// TIA Portal V18 program export: 1 tag tables, 8 data types, 17 data blocks, 20 code blocks (in call order from the OBs), 0 instance data blocks

VAR_GLOBAL   // PLC tag table "Default tag table"
   "AI11.01.01" AT %IW64 : Int;   // AHU NF Перепад тиску повітря (2.40)
   "AI11.01.02" AT %IW66 : Int;   // HS Вихід нагрівача (10.11)
   "DI11.01.01" AT %I0.0 : Bool;   // HS Режим роботи "Зима"
   "DI11.01.02" AT %I0.1 : Bool;   // HS Режим роботи "Авто"
   "DI11.01.03" AT %I0.2 : Bool;   // HS Відмова Котел 1
   "DI11.01.04" AT %I0.3 : Bool;   // HS Відмова Котел 2
   "DI11.01.05" AT %I0.4 : Bool;   // HS Норм. рівень води Котел 1 (10.80)
   "DI11.01.06" AT %I0.5 : Bool;   // HS Низький тиск Котел 1 (10.71)
   "DI11.01.07" AT %I0.6 : Bool;   // HS Високий тиск Котел 1 (10.72)
   "DI11.01.08" AT %I0.7 : Bool;   // HS Норм. рівень води Котел 2 (10.81)
   "DI11.01.09" AT %I1.0 : Bool;   // HS Низький тиск Котел 1 (10.73)
   "DI11.01.10" AT %I1.1 : Bool;   // HS Високий тиск Котел 1 (10.74)
   "DI11.01.11" AT %I1.2 : Bool;
   "DI11.01.12" AT %I1.3 : Bool;
   "DI11.01.13" AT %I1.4 : Bool;
   "DI11.01.14" AT %I1.5 : Bool;
   "DO11.01.01" AT %Q0.0 : Bool;
   "DO11.01.02" AT %Q0.1 : Bool;
   "DO11.01.03" AT %Q0.2 : Bool;
   "DO11.01.04" AT %Q0.3 : Bool;
   "DO11.01.05" AT %Q0.4 : Bool;
   "DO11.01.06" AT %Q0.5 : Bool;
   "DO11.01.07" AT %Q0.6 : Bool;
   "DO11.01.08" AT %Q0.7 : Bool;
   "DO11.01.09" AT %Q1.0 : Bool;
   "DO11.01.10" AT %Q1.1 : Bool;
   "AI11.02.01" AT %IW68 : Int;
   "AI11.02.02" AT %IW70 : Int;
   "AI11.02.03" AT %IW72 : Int;
   "AI11.02.04" AT %IW74 : Int;
   "AI11.02.05" AT %IW76 : Int;
   "AI11.02.06" AT %IW78 : Int;
   "AI11.02.07" AT %IW80 : Int;
   "AI11.02.08" AT %IW82 : Int;
   "AO11.03.01" AT %QW64 : Int;
   "AO11.03.02" AT %QW66 : Int;
   "AO11.03.03" AT %QW68 : Int;
   "AO11.03.04" AT %QW70 : Int;
   "DI11.04.01" AT %I2.0 : Bool;
   "DI11.04.02" AT %I2.1 : Bool;
   "DI11.04.03" AT %I2.2 : Bool;
   "DI11.04.04" AT %I2.3 : Bool;
   "DI11.04.05" AT %I2.4 : Bool;
   "DI11.04.06" AT %I2.5 : Bool;
   "DI11.04.07" AT %I2.6 : Bool;
   "DI11.04.08" AT %I2.7 : Bool;
   "DI11.04.09" AT %I3.0 : Bool;
   "DI11.04.10" AT %I3.1 : Bool;
   "DI11.04.11" AT %I3.2 : Bool;
   "DI11.04.12" AT %I3.3 : Bool;
   "DI11.04.13" AT %I3.4 : Bool;
   "DI11.04.14" AT %I3.5 : Bool;
   "DI11.04.15" AT %I3.6 : Bool;
   "DI11.04.16" AT %I3.7 : Bool;
   "DI11.05.01" AT %I4.0 : Bool;
   "DI11.05.02" AT %I4.1 : Bool;
   "DI11.05.03" AT %I4.2 : Bool;
   "DI11.05.04" AT %I4.3 : Bool;
   "DI11.05.05" AT %I4.4 : Bool;
   "DI11.05.06" AT %I4.5 : Bool;
   "DI11.05.07" AT %I4.6 : Bool;
   "DI11.05.08" AT %I4.7 : Bool;
   "DI11.05.09" AT %I5.0 : Bool;
   "DI11.05.10" AT %I5.1 : Bool;
   "DI11.05.11" AT %I5.2 : Bool;
   "DI11.05.12" AT %I5.3 : Bool;
   "DI11.05.13" AT %I5.4 : Bool;
   "DI11.05.14" AT %I5.5 : Bool;
   "DI11.05.15" AT %I5.6 : Bool;
   "DI11.05.16" AT %I5.7 : Bool;
   "DI11.06.01" AT %I6.0 : Bool;
   "DI11.06.02" AT %I6.1 : Bool;
   "DI11.06.03" AT %I6.2 : Bool;
   "DI11.06.04" AT %I6.3 : Bool;
   "DI11.06.05" AT %I6.4 : Bool;
   "DI11.06.06" AT %I6.5 : Bool;
   "DI11.06.07" AT %I6.6 : Bool;
   "DI11.06.08" AT %I6.7 : Bool;
   "DI11.06.09" AT %I7.0 : Bool;
   "DI11.06.10" AT %I7.1 : Bool;
   "DI11.06.11" AT %I7.2 : Bool;
   "DI11.06.12" AT %I7.3 : Bool;
   "DI11.06.13" AT %I7.4 : Bool;
   "DI11.06.14" AT %I7.5 : Bool;
   "DI11.06.15" AT %I7.6 : Bool;
   "DI11.06.16" AT %I7.7 : Bool;
   "DI11.07.01" AT %I8.0 : Bool;
   "DI11.07.02" AT %I8.1 : Bool;
   "DI11.07.03" AT %I8.2 : Bool;
   "DI11.07.04" AT %I8.3 : Bool;
   "DI11.07.05" AT %I8.4 : Bool;
   "DI11.07.06" AT %I8.5 : Bool;
   "DI11.07.07" AT %I8.6 : Bool;
   "DI11.07.08" AT %I8.7 : Bool;
   "DI11.07.09" AT %I9.0 : Bool;
   "DI11.07.10" AT %I9.1 : Bool;
   "DI11.07.11" AT %I9.2 : Bool;
   "DI11.07.12" AT %I9.3 : Bool;
   "DI11.07.13" AT %I9.4 : Bool;
   "DI11.07.14" AT %I9.5 : Bool;
   "DI11.07.15" AT %I9.6 : Bool;
   "DI11.07.16" AT %I9.7 : Bool;
   "DO11.08.01" AT %Q2.0 : Bool;
   "DO11.08.02" AT %Q2.1 : Bool;
   "DO11.08.03" AT %Q2.2 : Bool;
   "DO11.08.04" AT %Q2.3 : Bool;
   "DO11.08.05" AT %Q2.4 : Bool;
   "DO11.08.06" AT %Q2.5 : Bool;
   "DO11.08.07" AT %Q2.6 : Bool;
   "DO11.08.08" AT %Q2.7 : Bool;
   "DO11.08.09" AT %Q3.0 : Bool;
   "DO11.08.10" AT %Q3.1 : Bool;
   "DO11.08.11" AT %Q3.2 : Bool;
   "DO11.08.12" AT %Q3.3 : Bool;
   "DO11.08.13" AT %Q3.4 : Bool;
   "DO11.08.14" AT %Q3.5 : Bool;
   "DO11.08.15" AT %Q3.6 : Bool;
   "DO11.08.16" AT %Q3.7 : Bool;
   "DO11.09.01" AT %Q4.0 : Bool;
   "DO11.09.02" AT %Q4.1 : Bool;
   "DO11.09.03" AT %Q4.2 : Bool;
   "DO11.09.04" AT %Q4.3 : Bool;
   "DO11.09.05" AT %Q4.4 : Bool;
   "DO11.09.06" AT %Q4.5 : Bool;
   "DO11.09.07" AT %Q4.6 : Bool;
   "DO11.09.08" AT %Q4.7 : Bool;
   "DO11.09.09" AT %Q5.0 : Bool;
   "DO11.09.10" AT %Q5.1 : Bool;
   "DO11.09.11" AT %Q5.2 : Bool;
   "DO11.09.12" AT %Q5.3 : Bool;
   "DO11.09.13" AT %Q5.4 : Bool;
   "DO11.09.14" AT %Q5.5 : Bool;
   "DO11.09.15" AT %Q5.6 : Bool;
   "DO11.09.16" AT %Q5.7 : Bool;
   "AI11.10.01" AT %IW84 : Int;
   "AI11.10.02" AT %IW86 : Int;
   "AI11.10.03" AT %IW88 : Int;
   "AI11.10.04" AT %IW90 : Int;
   "AI11.10.05" AT %IW92 : Int;
   "AI11.10.06" AT %IW94 : Int;
   "AI11.10.07" AT %IW96 : Int;
   "AI11.10.08" AT %IW98 : Int;
   "AO11.11.01" AT %QW72 : Int;
   "AO11.11.02" AT %QW74 : Int;
   "AO11.11.03" AT %QW76 : Int;
   "AO11.11.04" AT %QW78 : Int;
END_VAR

TYPE "UDT_HWModulesMap"
// stored: IsFailsafeCompliant false
   STRUCT
      cRack : Byte;
      cModule : Byte;
      wLaddr1 : Word;
      wLaddr2 : Word;
      iDiagBuffer : USInt;
      iOwnState : UInt;
      wMaintenanceState : DWord;
      wComponentStateDetail : DWord;
      iOperatingState : UInt;
   END_STRUCT;
END_TYPE

TYPE "UDT_VirtModulesMap"
// stored: IsFailsafeCompliant false
   STRUCT
      cRack : Byte;
      cModule : Byte;
      iDiagBuffer : USInt;
      iOwnState : UInt;
   END_STRUCT;
END_TYPE

TYPE "UDT_AIadv"
// stored: IsFailsafeCompliant false
   STRUCT
      rValue : Real;   // Real value
      rMin : Real;   // Scale Min
      rMax : Real;   // Scale Max
      rCalibration : Real;
      iFuncSystemID : Byte := 0;
      iFuncVar : Byte := 0;
      rFilterSet : Real;   // Filter value
   END_STRUCT;
END_TYPE

TYPE "UDT_DIadv"
// stored: IsFailsafeCompliant false
   STRUCT
      xInput : Bool;
      xMemoryIn : Bool;   // Temp
      xMemoryOut : Bool;
      xInversion : Bool;   // DIs label for monitoring
      xOutput : Bool;   // Filtered value
      xtemp1 : Bool;
      xtemp2 : Bool;
      xtemp3 : Bool;
      cMemory : Byte := 0;
      iCounterOut : Int;
      iCounterIn : Int;   // Counter for DIs EDGE
      cFuncSystemID : Byte := 0;
      cFuncVar : Byte := 0;
      cDelayOnSec : Byte := 0;   // Temp
      cDelayOffSec : Byte := 0;   // Temp
   END_STRUCT;
END_TYPE

TYPE "UDT_RTDadv"
// stored: IsFailsafeCompliant false
   STRUCT
      rValue : Real;   // Real value
      rFilterSet : Real;   // Filter value
      rCalibration : Real;   // Scale Min
      rDiv : Real := 100.0;   // Scale Max
      cFuncSystemID : Byte := 0;
      cFuncVar : Byte := 0;
      iReserv : Int;
   END_STRUCT;
END_TYPE

TYPE "UDT_vAO"
// stored: IsFailsafeCompliant false
   STRUCT
      rInput : Real;   // Value for AO
      cMOA : Byte := 0;   // Mode Manual/Off/Auto
      cFuncSystemID : Byte := 0;
      cFuncVar : Byte := 0;
      cMemory : Byte := 0;
      rManOutput : Real;   // Manual output
      iOutput : Int;   // Output for DAC
   END_STRUCT;
END_TYPE

TYPE "UDT_vDI"
// stored: IsFailsafeCompliant false
   STRUCT
      xInput : Bool;
      xMemoryIn : Bool;   // Temp
      xMemoryOut : Bool;
      xInversion : Bool;   // DIs label for monitoring
      xOutput : Bool;   // Filtered value
      xtemp1 : Bool;
      xtemp2 : Bool;
      xtemp3 : Bool;
      cMemory : Byte := 0;
      iCounterOut : Int;
      iCounterIn : Int;   // Counter for DIs EDGE
      cFuncSystemID : Byte := 0;
      cFuncVar : Byte := 0;
      cDelayOnSec : Byte := 0;   // Temp
      cDelayOffSec : Byte := 0;   // Temp
   END_STRUCT;
END_TYPE

TYPE "UDT_vDO"
// stored: IsFailsafeCompliant false
   STRUCT
      xInput : Bool;   // Value for DO
      xOutput : Bool;   // Phisicl output
      xMemoryIn : Bool;   // Internal
      xInversion : Bool;
      xMemoryOut : Bool;
      xReserv3 : Bool;
      xReserv4 : Bool;
      xReserv5 : Bool;
      iCounterIn : Int;   // Counter
      iCounterOut : Int;
      iFuncSystemID : Byte := 0;
      iFuncVar : Byte := 0;
      cMOA : Byte;   // Mode Manual/Off/Auto
      cMemory : Byte;
   END_STRUCT;
END_TYPE

DATA_BLOCK "ActualHWAlarmsList"   // DB10001
{ S7_Optimized_Access := 'FALSE' }
VERSION : 0.1
// stored: AutoNumber false, DBAccessibleFromOPCUA true, IsOnlyStoredInLoadMemory false, IsWriteProtectedInAS false
   VAR
      iActiveFaults : DInt;
      iWriteIndex : Int;
      Log { S7_SetPoint := 'True'} : Array[0..99] of "UDT_HWAlarmEntry";
   END_VAR
BEGIN
END_DATA_BLOCK

DATA_BLOCK "HWModulesConf"   // DB10002
{ S7_Optimized_Access := 'TRUE' }
VERSION : 0.1
// stored: AutoNumber false, DBAccessibleFromOPCUA true, IsOnlyStoredInLoadMemory false, IsRetainMemResEnabled false, IsWriteProtectedInAS false, MemoryReserve 100
   VAR
      HW { S7_SetPoint := 'True'} : Array[1..14] of "UDT_HWModulesMap";
   END_VAR
BEGIN
   HW[1..8].cRack := 11;
   HW[9..14].cRack := 12;
   HW[1].cModule := 1;
   HW[2].cModule := 2;
   HW[3].cModule := 3;
   HW[4].cModule := 4;
   HW[5].cModule := 5;
   HW[6].cModule := 6;
   HW[7..8].cModule := 7;
   HW[9].cModule := 0;
   HW[10].cModule := 1;
   HW[11].cModule := 2;
   HW[12].cModule := 3;
   HW[13].cModule := 4;
   HW[14].cModule := 5;
   HW[1].wLaddr1 := 263;
   HW[2].wLaddr1 := 269;
   HW[3].wLaddr1 := 270;
   HW[4].wLaddr1 := 286;
   HW[5].wLaddr1 := 271;
   HW[6].wLaddr1 := 272;
   HW[7].wLaddr1 := 287;
   HW[8].wLaddr1 := 288;
   HW[9].wLaddr1 := 280;
   HW[10].wLaddr1 := 282;
   HW[11].wLaddr1 := 283;
   HW[12].wLaddr1 := 284;
   HW[13].wLaddr1 := 285;
   HW[14].wLaddr1 := 281;
   HW[1].wLaddr2 := 264;
END_DATA_BLOCK

DATA_BLOCK "HeatingPLC_vAO_Vars"   // DB11002
{ S7_Optimized_Access := 'FALSE' }
VERSION : 0.1
// stored: AutoNumber false, DBAccessibleFromOPCUA true, IsOnlyStoredInLoadMemory false, IsWriteProtectedInAS false
   VAR
      vAO1 { S7_SetPoint := 'True'} : "UDT_vAO";
      vAO2 { S7_SetPoint := 'True'} : "UDT_vAO";
      vAO3 { S7_SetPoint := 'True'} : "UDT_vAO";
      vAO4 { S7_SetPoint := 'True'} : "UDT_vAO";
      vAO5 { S7_SetPoint := 'True'} : "UDT_vAO";
      vAO6 { S7_SetPoint := 'True'} : "UDT_vAO";
      vAO7 { S7_SetPoint := 'True'} : "UDT_vAO";
      vAO8 { S7_SetPoint := 'True'} : "UDT_vAO";
   END_VAR
BEGIN
END_DATA_BLOCK

DATA_BLOCK "HeatingPLC_vDO_Vars"   // DB11004
{ S7_Optimized_Access := 'FALSE' }
VERSION : 0.1
// stored: AutoNumber false, DBAccessibleFromOPCUA true, IsOnlyStoredInLoadMemory false, IsWriteProtectedInAS false
   VAR
      vDO1 { S7_SetPoint := 'True'} : "UDT_vDO";
      vDO2 { S7_SetPoint := 'True'} : "UDT_vDO";
      vDO3 { S7_SetPoint := 'True'} : "UDT_vDO";
      vDO4 { S7_SetPoint := 'True'} : "UDT_vDO";
      vDO5 { S7_SetPoint := 'True'} : "UDT_vDO";
      vDO6 { S7_SetPoint := 'True'} : "UDT_vDO";
      vDO7 { S7_SetPoint := 'True'} : "UDT_vDO";
      vDO8 { S7_SetPoint := 'True'} : "UDT_vDO";
   END_VAR
BEGIN
END_DATA_BLOCK

DATA_BLOCK "SS1_710A1_8RTD_AI_Vars"   // DB11021
{ S7_Optimized_Access := 'FALSE' }
VERSION : 0.1
// stored: AutoNumber false, DBAccessibleFromOPCUA true, IsOnlyStoredInLoadMemory false, IsWriteProtectedInAS false
   VAR
      AI1 { S7_SetPoint := 'True'} : "UDT_RTDadv";   // Зовнішня температура (1.99)
      AI2 { S7_SetPoint := 'True'} : "UDT_RTDadv";   // AHU NF Темп. зв. теплоносія (2.57)
      AI3 { S7_SetPoint := 'True'} : "UDT_RTDadv";   // AHU NF Темп. припл. пов. (2.56)
      AI4 { S7_SetPoint := 'True'} : "UDT_RTDadv";   // AHU NF Кімнатна темп. (2.69)
      AI5 { S7_SetPoint := 'True'} : "UDT_RTDadv";   // HS Темп. под. теплоносія в колекторі (10.50)
      AI6 { S7_SetPoint := 'True'} : "UDT_RTDadv";   // Температура зв. теплоносія (8.66)
      AI7 { S7_SetPoint := 'True'} : "UDT_RTDadv";   // Темп. припл. пов. (8.68)
      AI8 { S7_SetPoint := 'True'} : "UDT_RTDadv";   // HS Темп. зв. теплоносія (10.92)
   END_VAR
BEGIN
   AI1.rValue := 26.03;
   AI1.rFilterSet := 0.0;
   AI1.rCalibration := 0.0;
   AI1.rDiv := 100.0;
   AI1.cFuncSystemID := 0;
   AI1.cFuncVar := 0;
   AI1.iReserv := 0;
   AI2.rValue := 3276.7;
   AI2.rFilterSet := 0.0;
   AI2.rCalibration := 0.0;
   AI2.rDiv := 10.0;
   AI2.cFuncSystemID := 2;
   AI2.cFuncVar := 0;
   AI2.iReserv := 0;
   AI3.rValue := 26.7;
   AI3.rFilterSet := 0.0;
   AI3.rCalibration := 0.0;
   AI3.rDiv := 100.0;
   AI3.cFuncSystemID := 16#01;
   AI3.cFuncVar := 16#04;
   AI3.iReserv := 0;
   AI4.rValue := 22.39;
   AI4.rFilterSet := 0.0;
   AI4.rCalibration := 0.0;
   AI4.rDiv := 100.0;
   AI4.cFuncSystemID := 16#03;
   AI4.cFuncVar := 16#04;
   AI4.iReserv := 0;
   AI5.rValue := 24.7;
   AI5.rFilterSet := 0.0;
   AI5.rCalibration := 0.0;
   AI5.rDiv := 10.0;
   AI5.cFuncSystemID := 16#0A;
   AI5.cFuncVar := 16#01;
   AI5.iReserv := 0;
   AI6.rValue := 61.78;
   AI6.rFilterSet := 0.0;
   AI6.rCalibration := 0.0;
   AI6.rDiv := 100.0;
   AI6.cFuncSystemID := 16#0E;
   AI6.cFuncVar := 16#01;
   AI6.iReserv := 0;
   AI7.rValue := 28.62;
   AI7.rFilterSet := 0.0;
   AI7.rCalibration := 0.0;
   AI7.rDiv := 100.0;
   AI7.cFuncSystemID := 16#0E;
   AI7.cFuncVar := 16#02;
   AI7.iReserv := 0;
   AI8.rValue := 21.31;
   AI8.rFilterSet := 0.0;
   AI8.rCalibration := 0.0;
   AI8.rDiv := 100.0;
   AI8.cFuncSystemID := 16#03;
   AI8.cFuncVar := 16#06;
   AI8.iReserv := 0;
END_DATA_BLOCK

DATA_BLOCK "SS1_730A1_4AO_AO_Vars"   // DB11041
{ S7_Optimized_Access := 'FALSE' }
VERSION : 0.1
// stored: AutoNumber false, DBAccessibleFromOPCUA true, IsOnlyStoredInLoadMemory false, IsWriteProtectedInAS false
   VAR
      AO1 { S7_SetPoint := 'True'} : "UDT_AOadv";   // AHU NF вихід нагрівача (2.58)
      AO2 { S7_SetPoint := 'True'} : "UDT_AOadv";   // AHU NF приточна/рециркуляційна заслінка (2.51/2.52)
      AO3 : "UDT_AOadv";   // Вихід нагрівача (8.67)
      AO4 : "UDT_AOadv";   // AHU NF витяжна заслінка (2.70)
   END_VAR
BEGIN
   AO1.cFuncSystemID := 1;
   AO1.cFuncVar := 2;
   AO2.cFuncSystemID := 1;
   AO2.cFuncVar := 3;
   AO3.cFuncSystemID := 3;
   AO3.cFuncVar := 2;
   AO4.cFuncSystemID := 1;
   AO4.cFuncVar := 4;
END_DATA_BLOCK

DATA_BLOCK "SS1_750A1_16DI_DI_Vars"   // DB11051
{ S7_Optimized_Access := 'FALSE' }
VERSION : 0.1
// stored: AutoNumber false, DBAccessibleFromOPCUA true, IsOnlyStoredInLoadMemory false, IsWriteProtectedInAS false
   VAR
      DI1 : "UDT_DIadv";   // Індикація живлення SS-1
      DI2 : "UDT_DIadv";   // HS Несправність системи опалення
      DI3 : "UDT_DIadv";   // HS Ін. 1- ст пальник К1
      DI4 : "UDT_DIadv";   // HS Ін. 2- ст пальник К1
      DI5 : "UDT_DIadv";   // Резерв
      DI6 : "UDT_DIadv";   // HS Аварія пальник К1
      DI7 : "UDT_DIadv";   // HS Ін. 1- ст пальник К2
      DI8 : "UDT_DIadv";   // HS Ін. 2- ст пальник К2
      DI9 { S7_SetPoint := 'True'} : "UDT_DIadv";   // HS Аварія пальник К2
      DI10 { S7_SetPoint := 'True'} : "UDT_DIadv";   // Резерв
      DI11 { S7_SetPoint := 'True'} : "UDT_DIadv";   // Резерв
      DI12 { S7_SetPoint := 'True'} : "UDT_DIadv";   // AHU NF Аварія ККБ
      DI13 { S7_SetPoint := 'True'} : "UDT_DIadv";   // AHU NF Ін. 1- ст. ККБ
      DI14 { S7_SetPoint := 'True'} : "UDT_DIadv";   // AHU NF Ін. 2- ст. ККБ
      DI15 { S7_SetPoint := 'True'} : "UDT_DIadv";   // Гот. роб. сист. обігр. дизельпроводу (10.211)
      DI16 { S7_SetPoint := 'True'} : "UDT_DIadv";   // AHU NF Гот. роб. обігр. пов. засл. (2.202)
   END_VAR
BEGIN
   DI3.cFuncSystemID := 10;
   DI3.cFuncVar := 25;
   DI4.cFuncSystemID := 10;
   DI4.cFuncVar := 26;
   DI5.cFuncSystemID := 10;
   DI5.cFuncVar := 27;
   DI6.cFuncSystemID := 100;
   DI6.cFuncVar := 11;
   DI7.cFuncSystemID := 100;
   DI7.cFuncVar := 12;
   DI8.cFuncSystemID := 10;
   DI8.cFuncVar := 24;
   DI9.cFuncSystemID := 10;
   DI9.cFuncVar := 22;
   DI10.xInversion := true;
   DI10.cFuncSystemID := 10;
   DI10.cFuncVar := 23;
   DI11.cFuncSystemID := 10;
   DI11.cFuncVar := 7;
   DI12.cFuncSystemID := 10;
   DI12.cFuncVar := 2;
   DI13.xInversion := true;
   DI13.cFuncSystemID := 10;
   DI13.cFuncVar := 3;
   DI14.cFuncSystemID := 10;
   DI14.cFuncVar := 5;
   DI15.xInversion := true;
   DI15.cFuncSystemID := 10;
   DI15.cFuncVar := 6;
END_DATA_BLOCK

DATA_BLOCK "SS1_754A1_16DI_DI_Vars"   // DB11061
{ S7_Optimized_Access := 'FALSE' }
VERSION : 0.1
// stored: AutoNumber false, DBAccessibleFromOPCUA true, IsOnlyStoredInLoadMemory false, IsWriteProtectedInAS false
   VAR
      DI1 : "UDT_DIadv";   // AHU NF Термостат загр. замерз. (2.50)
      DI2 : "UDT_DIadv";   // AHU NF Авто. режим пр. вент. (2.200)
      DI3 : "UDT_DIadv";   // AHU NF 1-шв. пр. вент. (2.200)
      DI4 : "UDT_DIadv";   // AHU NF 2-шв. пр. вент. (2.200)
      DI5 : "UDT_DIadv";   // AHU NF Тепл. реле. 1-шв. пр. вент. (2.200)
      DI6 : "UDT_DIadv";   // AHU NF Тепл. реле. 2-шв. пр. вент. (2.200)
      DI7 : "UDT_DIadv";   // AHU NF Несправність пр. вент. (2.200)
      DI8 : "UDT_DIadv";   // AHU NF Інд. сервісний вимикач. пр. вент. (2.200)
      DI9 { S7_SetPoint := 'True'} : "UDT_DIadv";   // AHU NF Несправність клиновий ркмінь пр. вент. (2.54)
      DI10 { S7_SetPoint := 'True'} : "UDT_DIadv";   // AHU NF Забруднення пр. фільтру (2.53)
      DI11 { S7_SetPoint := 'True'} : "UDT_DIadv";   // AHU NF Робота цирк. насос (2.201)
      DI12 { S7_SetPoint := 'True'} : "UDT_DIadv";   // AHU NF Авто режим цирк. насос (2.201)
      DI13 { S7_SetPoint := 'True'} : "UDT_DIadv";   // AHU NF Несправність цирк. насос (2.201)
      DI14 { S7_SetPoint := 'True'} : "UDT_DIadv";   // HS Робота вн. насос К1 (10.209)
      DI15 { S7_SetPoint := 'True'} : "UDT_DIadv";   // HS Перегрів вн. насос К1 (10.209) термоконтакт
      DI16 { S7_SetPoint := 'True'} : "UDT_DIadv";   // HS Робота вн. насос К2 (10.210)
   END_VAR
BEGIN
   DI1.cFuncSystemID := 100;
   DI1.cFuncVar := 1;
   DI2.cFuncSystemID := 100;
   DI2.cFuncVar := 3;
   DI5.cFuncSystemID := 100;
   DI5.cFuncVar := 5;
   DI6.cFuncSystemID := 100;
   DI6.cFuncVar := 6;
END_DATA_BLOCK

DATA_BLOCK "SS1_758A1_16DI_DI_Vars"   // DB11061
{ S7_Optimized_Access := 'FALSE' }
VERSION : 0.1
// stored: AutoNumber false, DBAccessibleFromOPCUA true, IsOnlyStoredInLoadMemory false, IsWriteProtectedInAS false
   VAR
      DI1 : "UDT_DIadv";   // HS Перегрів вн. наос К2 (10.20) термоконтакт
      DI2 : "UDT_DIadv";   // HS Авто режим насосів опалення (10.202+10.203)
      DI3 : "UDT_DIadv";   // HS Несправність насос опалення 1 (10.202)
      DI4 : "UDT_DIadv";   // HS Несправність насос опалення 2 (10.203)
      DI5 : "UDT_DIadv";   // Робота обігріву дизельпроводу
      DI6 : "UDT_DIadv";   // Резерв
      DI7 : "UDT_DIadv";   // Перегрів двигуна тепл. вентиляторів (8.215+8.216)
      DI8 : "UDT_DIadv";   // Робота тепл. вентиляторів (8.215+8.216)
      DI9 { S7_SetPoint := 'True'} : "UDT_DIadv";   // Термостат загр. замерз. (8.73)
      DI10 { S7_SetPoint := 'True'} : "UDT_DIadv";   // Термостат загр. замерз. (8.74)
      DI11 { S7_SetPoint := 'True'} : "UDT_DIadv";   // Несправність цирк. насос (8.217)
      DI12 { S7_SetPoint := 'True'} : "UDT_DIadv";   // Робота цирк. насос (8.217)
      DI13 { S7_SetPoint := 'True'} : "UDT_DIadv";   // Авто режим цирк. насос (8.217)
      DI14 { S7_SetPoint := 'True'} : "UDT_DIadv";   // Забруднення пр. фільтру (8.71)
      DI15 { S7_SetPoint := 'True'} : "UDT_DIadv";   // Забруднення пр. фільтру (8.72)
      DI16 { S7_SetPoint := 'True'} : "UDT_DIadv";   // HS Робота насосу опалення 1 (10.202)
   END_VAR
BEGIN
   DI1.cFuncSystemID := 100;
   DI1.cFuncVar := 1;
   DI2.cFuncSystemID := 100;
   DI2.cFuncVar := 3;
   DI5.cFuncSystemID := 100;
   DI5.cFuncVar := 5;
   DI6.cFuncSystemID := 100;
   DI6.cFuncVar := 6;
END_DATA_BLOCK

DATA_BLOCK "SS1_762A1_16DI_DI_Vars"   // DB11061
{ S7_Optimized_Access := 'FALSE' }
VERSION : 0.1
// stored: AutoNumber false, DBAccessibleFromOPCUA true, IsOnlyStoredInLoadMemory false, IsWriteProtectedInAS false
   VAR
      DI1 : "UDT_DIadv";   // HS Робота насосу опалення 2 (10.203)
      DI2 : "UDT_DIadv";   // Резерв
      DI3 : "UDT_DIadv";   // Резерв
      DI4 : "UDT_DIadv";   // Резерв
      DI5 : "UDT_DIadv";   // Резерв
      DI6 : "UDT_DIadv";   // Резерв
      DI7 : "UDT_DIadv";   // Резерв
      DI8 : "UDT_DIadv";   // Резерв
      DI9 { S7_SetPoint := 'True'} : "UDT_DIadv";   // Резерв
      DI10 { S7_SetPoint := 'True'} : "UDT_DIadv";   // Резерв
      DI11 { S7_SetPoint := 'True'} : "UDT_DIadv";   // Резерв
      DI12 { S7_SetPoint := 'True'} : "UDT_DIadv";   // Резерв
      DI13 { S7_SetPoint := 'True'} : "UDT_DIadv";   // Резерв
      DI14 { S7_SetPoint := 'True'} : "UDT_DIadv";   // Резерв
      DI15 { S7_SetPoint := 'True'} : "UDT_DIadv";   // Резерв
      DI16 { S7_SetPoint := 'True'} : "UDT_DIadv";   // Резерв
   END_VAR
BEGIN
   DI1.cFuncSystemID := 100;
   DI1.cFuncVar := 1;
   DI2.cFuncSystemID := 100;
   DI2.cFuncVar := 3;
   DI5.cFuncSystemID := 100;
   DI5.cFuncVar := 5;
   DI6.cFuncSystemID := 100;
   DI6.cFuncVar := 6;
END_DATA_BLOCK

DATA_BLOCK "SS1_770A1_16DO_DO_Vars"   // DB11072
{ S7_Optimized_Access := 'FALSE' }
VERSION : 0.1
// stored: AutoNumber false, DBAccessibleFromOPCUA true, IsOnlyStoredInLoadMemory false, IsWriteProtectedInAS false
   VAR
      DO1 { S7_SetPoint := 'True'} : "UDT_DOadv";   // Резерв
      DO2 { S7_SetPoint := 'True'} : "UDT_DOadv";   // Резерв
      DO3 { S7_SetPoint := 'True'} : "UDT_DOadv";   // Вкл. тепл. вент (8.x)
      DO4 { S7_SetPoint := 'True'} : "UDT_DOadv";   // HS Вкл. насос (10.203)
      DO5 { S7_SetPoint := 'True'} : "UDT_DOadv";   // HS Вкл. насос (10.202)
      DO6 { S7_SetPoint := 'True'} : "UDT_DOadv";   // HS Дозвіл на роботу пальник 1- ст. К1
      DO7 { S7_SetPoint := 'True'} : "UDT_DOadv";   // HS Дозвіл на роботу пальник 2- ст. К1
      DO8 { S7_SetPoint := 'True'} : "UDT_DOadv";   // AHU NF Вкл. цирк. насос (2.202)
      DO9 { S7_SetPoint := 'True'} : "UDT_DOadv";   // AHU NF Дозвіл на роботу 1- ст. ККБ
      DO10 { S7_SetPoint := 'True'} : "UDT_DOadv";   // AHU NF Дозвіл на роботу 2- ст. ККБ
      DO11 { S7_SetPoint := 'True'} : "UDT_DOadv";   // AHU NF Дозвіл на роботу 3- ст. ККБ
      DO12 { S7_SetPoint := 'True'} : "UDT_DOadv";   // AHU NF Дозвіл на роботу 4- ст. ККБ
      DO13 { S7_SetPoint := 'True'} : "UDT_DOadv";   // AHU NF Вкл. 1- шв. пр. вент. (2.200)
      DO14 { S7_SetPoint := 'True'} : "UDT_DOadv";   // AHU NF Вкл. 2- шв. пр. вент. (2.200)
      DO15 { S7_SetPoint := 'True'} : "UDT_DOadv";   // HS Дозвіл на роботу пальник 1- ст. К2
      DO16 { S7_SetPoint := 'True'} : "UDT_DOadv";   // HS Дозвіл на роботу пальник 2- ст. К2
   END_VAR
BEGIN
   DO1.iFuncSystemID := 10;
   DO1.iFuncVar := 10;
   DO2.iFuncSystemID := 10;
   DO2.iFuncVar := 11;
   DO3.iFuncSystemID := 10;
   DO3.iFuncVar := 12;
   DO4.iFuncSystemID := 100;
   DO4.iFuncVar := 1;
   DO5.iFuncSystemID := 100;
   DO5.iFuncVar := 5;
   DO6.iFuncSystemID := 100;
   DO6.iFuncVar := 3;
   DO7.iFuncSystemID := 10;
   DO7.iFuncVar := 5;
   DO8.iFuncSystemID := 10;
   DO8.iFuncVar := 6;
   DO9.iFuncSystemID := 10;
   DO9.iFuncVar := 13;
   DO14.iFuncSystemID := 1;
   DO14.iFuncVar := 1;
   DO14.cMOA := 1;
   DO15.iFuncSystemID := 1;
   DO16.iFuncSystemID := 1;
   DO16.iFuncVar := 3;
END_DATA_BLOCK

DATA_BLOCK "SS1_774A1_16DO_DO_Vars"   // DB11072
{ S7_Optimized_Access := 'FALSE' }
VERSION : 0.1
// stored: AutoNumber false, DBAccessibleFromOPCUA true, IsOnlyStoredInLoadMemory false, IsWriteProtectedInAS false
   VAR
      DO1 { S7_SetPoint := 'True'} : "UDT_DOadv";   // HS Вкл. вн. насос К1 (10.209)
      DO2 { S7_SetPoint := 'True'} : "UDT_DOadv";   // HS Вкл. вн. насос К2 (10.210)
      DO3 { S7_SetPoint := 'True'} : "UDT_DOadv";   // Резерв
      DO4 { S7_SetPoint := 'True'} : "UDT_DOadv";   // HS Дозвіл на роботу котлів
      DO5 { S7_SetPoint := 'True'} : "UDT_DOadv";   // AHU NF Вкл. обігріву пов. засл. (2.202)
      DO6 { S7_SetPoint := 'True'} : "UDT_DOadv";   // Вкл. обігріву дизельпровода (10.211)
      DO7 { S7_SetPoint := 'True'} : "UDT_DOadv";   // Вкл. системи кондиціювання (7.208 + 7.210)
      DO8 { S7_SetPoint := 'True'} : "UDT_DOadv";   // Вкл. тепл. вентилятор (8.215 + 8.216)
      DO9 { S7_SetPoint := 'True'} : "UDT_DOadv";   // Вкл. цирк. насос (8.217)
      DO10 { S7_SetPoint := 'True'} : "UDT_DOadv";   // Резерв
      DO11 { S7_SetPoint := 'True'} : "UDT_DOadv";   // Резерв
      DO12 { S7_SetPoint := 'True'} : "UDT_DOadv";   // Резерв
      DO13 { S7_SetPoint := 'True'} : "UDT_DOadv";   // Резерв
      DO14 { S7_SetPoint := 'True'} : "UDT_DOadv";   // Резерв
      DO15 { S7_SetPoint := 'True'} : "UDT_DOadv";   // Резерв
      DO16 { S7_SetPoint := 'True'} : "UDT_DOadv";   // Резерв
   END_VAR
BEGIN
   DO1.iFuncSystemID := 10;
   DO1.iFuncVar := 10;
   DO2.iFuncSystemID := 10;
   DO2.iFuncVar := 11;
   DO3.iFuncSystemID := 10;
   DO3.iFuncVar := 12;
   DO4.iFuncSystemID := 100;
   DO4.iFuncVar := 1;
   DO5.iFuncSystemID := 100;
   DO5.iFuncVar := 5;
   DO6.iFuncSystemID := 100;
   DO6.iFuncVar := 3;
   DO7.iFuncSystemID := 10;
   DO7.iFuncVar := 5;
   DO8.iFuncSystemID := 10;
   DO8.iFuncVar := 6;
   DO9.iFuncSystemID := 10;
   DO9.iFuncVar := 13;
   DO14.iFuncSystemID := 1;
   DO14.iFuncVar := 1;
   DO14.cMOA := 1;
   DO15.iFuncSystemID := 1;
   DO16.iFuncSystemID := 1;
   DO16.iFuncVar := 3;
END_DATA_BLOCK

DATA_BLOCK "SS1_780A1_8xAI_AI_Vars"   // DB11031
{ S7_Optimized_Access := 'FALSE' }
VERSION : 0.1
// stored: AutoNumber false, DBAccessibleFromOPCUA true, IsOnlyStoredInLoadMemory false, IsWriteProtectedInAS false
   VAR
      AI1 { S7_SetPoint := 'True'} : "UDT_AIadv";   // HS Температура в прим. котельні (10.02)
      AI2 { S7_SetPoint := 'True'} : "UDT_AIadv";   // 4-wire
      AI3 { S7_SetPoint := 'True'} : "UDT_AIadv";   // HS Температура зв. теплоносія (10.12)
      AI4 { S7_SetPoint := 'True'} : "UDT_AIadv";   // 4-wire
      AI5 { S7_SetPoint := 'True'} : "UDT_AIadv";   // HS Температура подачі теплоносія (10.13)
      AI6 { S7_SetPoint := 'True'} : "UDT_AIadv";   // 4-wire
      AI7 { S7_SetPoint := 'True'} : "UDT_AIadv";   // Резерв
      AI8 { S7_SetPoint := 'True'} : "UDT_AIadv";   // Резерв
   END_VAR
BEGIN
   AI1.rValue := 0.3255208;
   AI1.rMin := 0.0;
   AI1.rMax := 1000.0;
   AI1.rCalibration := 0.0;
   AI1.iFuncSystemID := 16#00;
   AI1.iFuncVar := 16#00;
   AI1.rFilterSet := 0.0;
   AI2.rValue := 1.808449;
   AI2.rMin := 0.0;
   AI2.rMax := 1000.0;
   AI2.rCalibration := 0.0;
   AI2.iFuncSystemID := 16#00;
   AI2.iFuncVar := 16#00;
   AI2.rFilterSet := 0.0;
   AI3.rValue := 3.616898E-05;
   AI3.rMin := 0.0;
   AI3.rMax := 0.0;
   AI3.rCalibration := 0.0;
   AI3.iFuncSystemID := 16#00;
   AI3.iFuncVar := 16#00;
   AI3.rFilterSet := 0.0;
   AI4.rValue := 0.0003255208;
   AI4.rMin := 0.0;
   AI4.rMax := 0.0;
   AI4.rCalibration := 0.0;
   AI4.iFuncSystemID := 16#00;
   AI4.iFuncVar := 16#00;
   AI4.rFilterSet := 0.0;
   AI5.rValue := 6.04022;
   AI5.rMin := 0.0;
   AI5.rMax := 1000.0;
   AI5.rCalibration := 0.0;
   AI5.iFuncSystemID := 16#01;
   AI5.iFuncVar := 16#0A;
   AI5.rFilterSet := 0.0;
   AI6.rValue := 17.15549;
   AI6.rMin := 0.0;
   AI6.rMax := 15.0;
   AI6.rCalibration := 0.0;
   AI6.iFuncSystemID := 16#01;
   AI6.iFuncVar := 16#07;
   AI6.rFilterSet := 0.0;
   AI7.rValue := 29.49942;
   AI7.rMin := 0.0;
   AI7.rMax := 100.0;
   AI7.rCalibration := 0.0;
   AI7.iFuncSystemID := 16#00;
   AI7.iFuncVar := 16#00;
   AI7.rFilterSet := 0.0;
   AI8.rValue := 0.07957176;
   AI8.rMin := 0.0;
   AI8.rMax := 100.0;
   AI8.rCalibration := 0.0;
   AI8.iFuncSystemID := 16#00;
   AI8.iFuncVar := 16#00;
   AI8.rFilterSet := 0.0;
END_DATA_BLOCK

DATA_BLOCK "SS1_784A1_4AO_AO_Vars"   // DB11041
{ S7_Optimized_Access := 'FALSE' }
VERSION : 0.1
// stored: AutoNumber false, DBAccessibleFromOPCUA true, IsOnlyStoredInLoadMemory false, IsWriteProtectedInAS false
   VAR
      AO1 { S7_SetPoint := 'True'} : "UDT_AOadv";   // HS Вихід нагрівача контуру опалення (10.11)
      AO2 { S7_SetPoint := 'True'} : "UDT_AOadv";   // Резерв
      AO3 : "UDT_AOadv";   // Резерв
      AO4 : "UDT_AOadv";   // Резерв
   END_VAR
BEGIN
   AO1.cFuncSystemID := 1;
   AO1.cFuncVar := 2;
   AO2.cFuncSystemID := 1;
   AO2.cFuncVar := 3;
   AO3.cFuncSystemID := 3;
   AO3.cFuncVar := 2;
   AO4.cFuncSystemID := 1;
   AO4.cFuncVar := 4;
END_DATA_BLOCK

DATA_BLOCK "SS1_CPU1214_AI_Vars"   // DB11011
{ S7_Optimized_Access := 'FALSE' }
VERSION : 0.1
// stored: AutoNumber false, DBAccessibleFromOPCUA true, IsOnlyStoredInLoadMemory false, IsWriteProtectedInAS false
   VAR
      AI1 { S7_SetPoint := 'True'} : "UDT_AIadv";   // AHU NF Перепад тиску повітря (2.40)
      AI2 { S7_SetPoint := 'True'} : "UDT_AIadv";   // HS Вихід нагрівача (10.11)
   END_VAR
BEGIN
   AI1.rValue := 368.9236;
   AI1.rMin := 0.0;
   AI1.rMax := 50000.0;
   AI1.rCalibration := 0.0;
   AI1.iFuncSystemID := 2;
   AI1.iFuncVar := 2;
   AI1.rFilterSet := 0.0;
   AI2.rValue := 0.0;
   AI2.rMin := 0.0;
   AI2.rMax := 0.0;
   AI2.rCalibration := 0.0;
   AI2.iFuncSystemID := 10;
   AI2.iFuncVar := 7;
   AI2.rFilterSet := 0.0;
END_DATA_BLOCK

DATA_BLOCK "SS1_CPU1214_DI_Vars"   // DB11013
{ S7_Optimized_Access := 'FALSE' }
VERSION : 0.1
// stored: AutoNumber false, DBAccessibleFromOPCUA true, IsOnlyStoredInLoadMemory false, IsWriteProtectedInAS false
   VAR
      DI1 : "UDT_DIadv";   // HS Режим роботи "Зима"
      DI2 : "UDT_DIadv";   // HS Режим роботи "Авто"
      DI3 : "UDT_DIadv";   // HS Відмова Котел 1
      DI4 : "UDT_DIadv";   // HS Відмова Котел 2
      DI5 : "UDT_DIadv";   // HS Норм. рівень води Котел 1 (10.80)
      DI6 : "UDT_DIadv";   // HS Низький тиск Котел 1 (10.71)
      DI7 { S7_SetPoint := 'True'} : "UDT_DIadv";   // HS Високий тиск Котел 1 (10.72)
      DI8 { S7_SetPoint := 'True'} : "UDT_DIadv";   // HS Норм. рівень води Котел 2 (10.81)
      DI9 { S7_SetPoint := 'True'} : "UDT_DIadv";   // HS Низький тиск Котел 1 (10.73)
      DI10 { S7_SetPoint := 'True'} : "UDT_DIadv";   // HS Високий тиск Котел 1 (10.74)
      DI11 { S7_SetPoint := 'True'} : "UDT_DIadv";   // Резерв
      DI12 { S7_SetPoint := 'True'} : "UDT_DIadv";   // Резерв
      DI13 { S7_SetPoint := 'True'} : "UDT_DIadv";   // Резерв
      DI14 { S7_SetPoint := 'True'} : "UDT_DIadv";   // Резерв
   END_VAR
BEGIN
   DI1.cFuncSystemID := 3;
   DI1.cFuncVar := 19;
   DI2.cFuncSystemID := 3;
   DI2.cFuncVar := 8;
   DI3.cFuncSystemID := 3;
   DI3.cFuncVar := 9;
   DI4.cFuncSystemID := 3;
   DI4.cFuncVar := 20;
   DI5.cFuncSystemID := 3;
   DI5.cFuncVar := 7;
   DI6.cFuncSystemID := 3;
   DI6.cFuncVar := 21;
   DI8.cFuncSystemID := 10;
   DI8.cFuncVar := 41;
   DI9.cFuncSystemID := 10;
   DI9.cFuncVar := 43;
   DI10.cFuncSystemID := 3;
   DI10.cFuncVar := 16;
   DI11.cFuncSystemID := 0;
   DI11.cFuncVar := 0;
   DI12.cFuncSystemID := 0;
   DI12.cFuncVar := 0;
   DI13.cFuncSystemID := 0;
   DI13.cFuncVar := 0;
END_DATA_BLOCK

DATA_BLOCK "SS1_CPU1214_DO_Vars"   // DB11014
{ S7_Optimized_Access := 'FALSE' }
VERSION : 0.1
// stored: AutoNumber false, DBAccessibleFromOPCUA true, IsOnlyStoredInLoadMemory false, IsWriteProtectedInAS false
   VAR
      DO1 { S7_SetPoint := 'True'} : "UDT_DOadv";   // Резерв
      DO2 { S7_SetPoint := 'True'} : "UDT_DOadv";   // Резерв
      DO3 { S7_SetPoint := 'True'} : "UDT_DOadv";   // Резерв
      DO4 { S7_SetPoint := 'True'} : "UDT_DOadv";   // Резерв
      DO5 { S7_SetPoint := 'True'} : "UDT_DOadv";   // Резерв
      DO6 : "UDT_DOadv";   // Резерв
      DO7 { S7_SetPoint := 'True'} : "UDT_DOadv";   // Резерв
      DO8 { S7_SetPoint := 'True'} : "UDT_DOadv";   // Резерв
      DO9 { S7_SetPoint := 'True'} : "UDT_DOadv";   // Резерв
      DO10 { S7_SetPoint := 'True'} : "UDT_DOadv";   // Резерв
   END_VAR
BEGIN
END_DATA_BLOCK

ORGANIZATION_BLOCK "Main"   // OB1, LAD, ProgramCycle
TITLE = "Main Program Sweep (Cycle)"
{ S7_Optimized_Access := 'TRUE' }
VERSION : 0.1
// stored: AutoNumber true, IsIECCheckEnabled false, SetENOAutomatically false
   VAR_INPUT
      Initial_Call : Bool;   // Initial call of this OB
      Remanence : Bool;   // =True, if remanent data are available
   END_VAR
BEGIN
END_ORGANIZATION_BLOCK

FUNCTION "AIadv" : Void   // FC10013, FBD
{ S7_Optimized_Access := 'TRUE' }
VERSION : 0.1
// stored: AutoNumber false, IsIECCheckEnabled false, SetENOAutomatically false, UDAEnableTagReadback false
   VAR_INPUT
      iInput : Int;
      rFilterValue : Real;
      rMin : Real;
      rMax : Real;
      rCalibration : Real;
   END_VAR
   VAR_OUTPUT
      rOutput : Real;
   END_VAR
   VAR_TEMP
      rNorm : Real;
      rScaled : Real;
      rOut_real : Real;
   END_VAR
   VAR CONSTANT
      iRawMin : Int := 0;
      iRawMax : Int := 27648;
   END_VAR
BEGIN

REGION Network 1 (SCL)
   #rNorm := NORM_X(
                    MIN := #iRawMin,
                    VALUE := #iInput,
                    MAX := #iRawMax);
END_REGION

REGION Network 2 (SCL)
   #rScaled := SCALE_X(
                       MIN := #rMin,
                       VALUE := #rNorm,
                       MAX := #rMax);
END_REGION

REGION Network 3 (SCL): // --- Обмеження межами ---
   IF #rScaled < #rMin THEN
       #rScaled := #rMin;
   ELSIF #rScaled > #rMax THEN
       #rScaled := #rMax;
   END_IF;
END_REGION

REGION Network 4 (SCL): // --- Калібрування (зсув) ---
   #rOutput := #rScaled + #rCalibration;
END_REGION

REGION Network 5 (SCL): // --- Підготовка коеф. фільтра ---
   // rFilterSet = 1.0 → фільтр «прозорий» (швидка реакція, без згладжування).
   // 
   // rFilterSet = 0.1…0.3 → м’яке згладжування.
   // 
   // rFilterSet = 0.0 → вихід «заморожений».
   // --- Підготовка коеф. фільтра ---
   //rAlpha := rFilterSet;/
   //IF rAlpha < 0.0 THEN
   //    rAlpha := 0.0;
   //END_IF;
   //IF rAlpha > 1.0 THEN
   //    rAlpha := 1.0;
   //END_IF;

   // --- Ініціалізація ---
   //IF xInit THEN
   //    rY := rScaledRaw;/
   //    xInit := FALSE;
   //END_IF;

   // --- Фільтр: y = y + α*(x - y) ---
   //rY := rY + rAlpha * (rScaledRaw - rY);

   // --- Вихід ---
   //#rOutput := rY;
END_REGION
END_FUNCTION

FUNCTION "AOadv" : Void   // FC10012, FBD
{ S7_Optimized_Access := 'TRUE' }
VERSION : 0.1
// stored: AutoNumber false, IsIECCheckEnabled false, SetENOAutomatically false, UDAEnableTagReadback false
   VAR_INPUT
      rInput : Real;   // 0 to 100
      cM0A : Byte;   // 0-direct / 1-reverse / 0-outp_off / 1- out=MAN_OUTPUT /2 -out=input
      rManOutput : Real;
   END_VAR
   VAR_OUTPUT
      iOutput : Int;
   END_VAR
   VAR_TEMP
      rOut : Real;
      rOutScaled : Real;
      rManOutputTemp : Real;
      iManOutputTemp : Int;
   END_VAR
   VAR CONSTANT
      iRawMin : Int := 0;
      iRawMax : Int := 27648;
   END_VAR
BEGIN

REGION Network 1 (SCL): // --- Вибір режиму ---
   // --- Вибір режиму ---
   CASE #cM0A OF
       0: // Off
           #rOut := 0.0;
       1: // Manual
           #rOut := #rManOutput;
       2: // Auto
           #rOut := #rInput;
       ELSE
           #rOut := 0.0; // захист від некоректних значень
   END_CASE;
END_REGION

REGION Network 2 (SCL): // --- Обмеження в межах 0.0…100.0 ---
   // --- Обмеження в межах 0.0…100.0 ---
   IF #rOut < 0.0 THEN
       #rOut := 0.0;
   ELSIF
       #rOut > 100.0 THEN
       #rOut := 100.0;
   END_IF;
END_REGION

REGION Network 3 (SCL)
   #rOutScaled := (#rOut * 27648.0) / 100;
END_REGION

REGION Network 4 (SCL)
   IF #rOutScaled < 0.0 THEN
       #rOutScaled := 0.0;
   ELSIF
       #rOutScaled > 27648.0 THEN
       #rOutScaled := 27648.0;
   END_IF;
END_REGION

REGION Network 5 (SCL)
   #iOutput := REAL_TO_INT(#rOutScaled + 0.5);
END_REGION
END_FUNCTION

FUNCTION "DOadv" : Void   // FC10009, LAD
{ S7_Optimized_Access := 'TRUE' }
VERSION : 0.1
// stored: AutoNumber false, IsIECCheckEnabled false, SetENOAutomatically false, UDAEnableTagReadback false
   VAR_INPUT
      xInput : Bool;
      xInversion : Bool;   // 0-direct / 1-reverse
      cMOA : Byte;
   END_VAR
   VAR_OUTPUT
      xOutput : Bool;
   END_VAR
   VAR_IN_OUT
      xMemoryOut : Bool;
      xMemoryIn : Bool;
      cMemory : Byte;
      iCounterIn : Int;
      iCounterOut : Int;
   END_VAR
   VAR_TEMP
      InOut_1 : Bool;
   END_VAR
BEGIN

REGION Network 1 (SCL)
   CASE #cMOA OF
       0: // OFF
           #xOutput := FALSE;

       1: // MANUAL
           #xOutput := TRUE;

       2: // AUTO
           #xOutput :=#xInput;

   ELSE
       #xOutput := FALSE;
   END_CASE;
END_REGION

REGION Network 2 (SCL)
   IF #xInversion THEN
       #xOutput := NOT #xOutput;
   END_IF;
END_REGION

REGION Network 3 (SCL)
   IF (#xMemoryIn XOR #xInput) THEN
       IF #iCounterIn > 30000 THEN
           #iCounterIn := 5;
       ELSE
           #iCounterIn := #iCounterIn + 1;
       END_IF;
   END_IF;
   #xMemoryIn := #xInput;
END_REGION

REGION Network 4 (SCL)
   IF (#xMemoryOut XOR #xOutput) THEN
       IF #iCounterOut > 30000 THEN
           #iCounterOut := 5;
       ELSE
           #iCounterOut := #iCounterOut + 1;
       END_IF;
   END_IF;
   #xMemoryOut := #xOutput;
END_REGION
END_FUNCTION

FUNCTION "DObasic" : Void   // FC10004, FBD
{ S7_Optimized_Access := 'TRUE' }
VERSION : 0.1
// stored: AutoNumber false, IsIECCheckEnabled false, SetENOAutomatically false, UDAEnableTagReadback false
   VAR_INPUT
      xInput : Bool;
      cM0A : Byte;   // 0-direct / 1-reverse / 0-outp_off / 1- aut=1 /2 -out=input
   END_VAR
   VAR_OUTPUT
      iCounter : Int;
      xOutput : Bool;
   END_VAR
   VAR_IN_OUT
      Bit_Count_1 : Bool;
   END_VAR
   VAR_TEMP
      cM0A_0 : Bool;
      cM0A_1 : Bool;
      cM0A_2 : Bool;
   END_VAR
   VAR CONSTANT
      bit_count : Bool;
   END_VAR
   VAR_TEMP   // added for the SCL form of the ladder/FBD networks
      _w1 : Bool;
   END_VAR
BEGIN

REGION Network 1
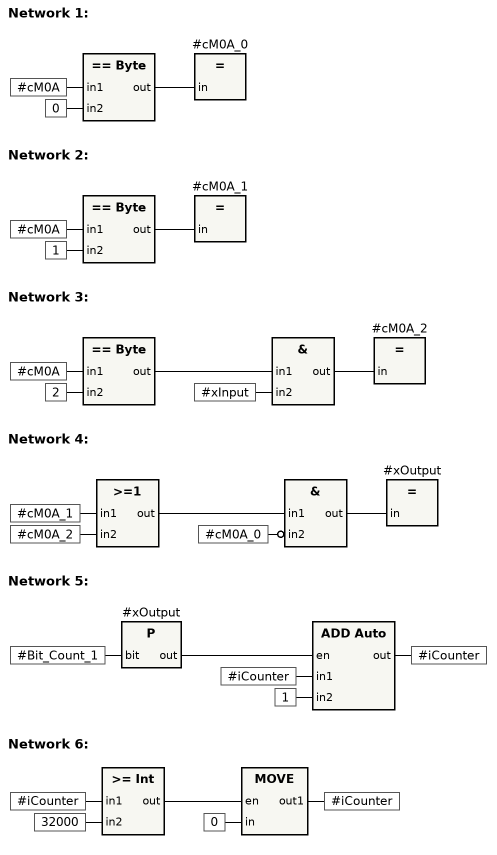
   #cM0A_0 := #cM0A = 0;
END_REGION

REGION Network 2
   #cM0A_1 := #cM0A = 1;
END_REGION

REGION Network 3
   #cM0A_2 := (#cM0A = 2) AND #xInput;
END_REGION

REGION Network 4
   #xOutput := (#cM0A_1 OR #cM0A_2) AND NOT #cM0A_0;
END_REGION

REGION Network 5
   #_w1 := #xOutput AND NOT #Bit_Count_1;   // rising edge of #xOutput
   #Bit_Count_1 := #xOutput;
   IF #_w1 THEN #iCounter := #iCounter + 1; END_IF;
END_REGION

REGION Network 6
   IF #iCounter >= 32000 THEN #iCounter := 0; END_IF;
END_REGION
END_FUNCTION

FUNCTION "RTDadv" : Void   // FC10015, FBD
{ S7_Optimized_Access := 'TRUE' }
VERSION : 0.1
// stored: AutoNumber false, IsIECCheckEnabled false, SetENOAutomatically false, UDAEnableTagReadback false
   VAR_INPUT
      iInput : Int;
      rFilterValue : Real;
      rCalibration : Real;
      rDiv : Real;
   END_VAR
   VAR_OUTPUT
      rOutput : Real;
   END_VAR
   VAR_TEMP
      rTemp : Real;
   END_VAR
   VAR CONSTANT
      rMin : Real := -50.0;
      rMax : Real := 150.0;
   END_VAR
BEGIN

REGION Network 1 (SCL)
   #rTemp := INT_TO_REAL(#iInput);
END_REGION

REGION Network 2 (SCL)
   #rTemp := #rTemp / #rDiv;
END_REGION

REGION Network 3 (SCL)
   #rTemp := #rTemp + #rCalibration;
END_REGION

REGION Network 4 (SCL): Filter
END_REGION

REGION Network 5 (SCL): Output
   //xValid := xDiagOK AND (rTempCalc > -250.0) AND (rTempCalc < 1000.0);
   //IF xValid THEN
   //    rTempC := rTempCalc;
   //END_IF;
   //
   #rOutput := #rTemp;
END_REGION
END_FUNCTION

FUNCTION "RTDbasic" : Void   // FC10006, FBD
{ S7_Optimized_Access := 'TRUE' }
VERSION : 0.1
// stored: AutoNumber false, IsIECCheckEnabled false, SetENOAutomatically false, UDAEnableTagReadback false
   VAR_INPUT
      iInput : Int;
      rFilterValue : Real;
      rCalibration : Real;
      rDiv : Real;
   END_VAR
   VAR_OUTPUT
      rOutput : Real;
   END_VAR
BEGIN
END_FUNCTION

FUNCTION "HeatingPLC_vIO" : Void   // FC11001, LAD
{ S7_Optimized_Access := 'FALSE' }
VERSION : 0.1
// stored: AutoNumber false, IsIECCheckEnabled false, SetENOAutomatically false, UDAEnableTagReadback false
BEGIN

REGION Network 1
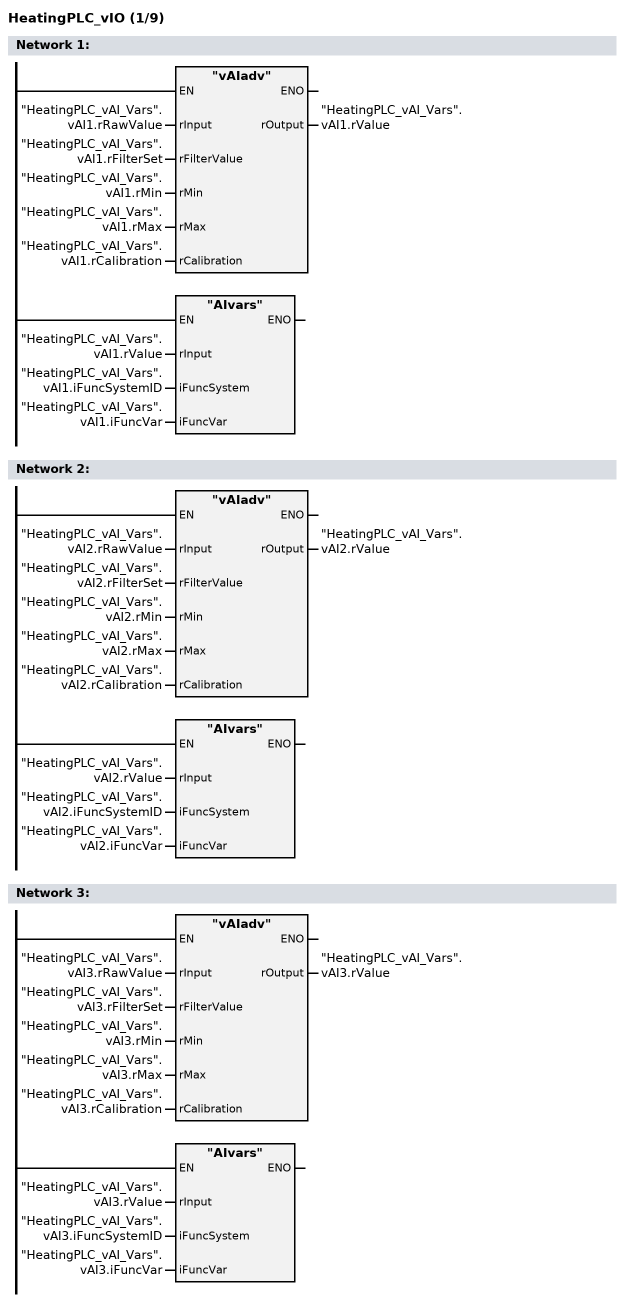
   RUNG wire#powerrail
      "vAIadv"(rInput := "HeatingPLC_vAI_Vars".vAI1.rRawValue, rFilterValue := "HeatingPLC_vAI_Vars".vAI1.rFilterSet, rMin := "HeatingPLC_vAI_Vars".vAI1.rMin, rMax := "HeatingPLC_vAI_Vars".vAI1.rMax, rCalibration := "HeatingPLC_vAI_Vars".vAI1.rCalibration, rOutput => "HeatingPLC_vAI_Vars".vAI1.rValue)
   END_RUNG
   RUNG wire#powerrail
      "AIvars"(rInput := "HeatingPLC_vAI_Vars".vAI1.rValue, iFuncSystem := "HeatingPLC_vAI_Vars".vAI1.iFuncSystemID, iFuncVar := "HeatingPLC_vAI_Vars".vAI1.iFuncVar)
   END_RUNG
   // the same network as SCL:
   "vAIadv"(rInput := "HeatingPLC_vAI_Vars".vAI1.rRawValue,
            rFilterValue := "HeatingPLC_vAI_Vars".vAI1.rFilterSet,
            rMin := "HeatingPLC_vAI_Vars".vAI1.rMin,
            rMax := "HeatingPLC_vAI_Vars".vAI1.rMax,
            rCalibration := "HeatingPLC_vAI_Vars".vAI1.rCalibration,
            rOutput => "HeatingPLC_vAI_Vars".vAI1.rValue);
   "AIvars"(rInput := "HeatingPLC_vAI_Vars".vAI1.rValue,
            iFuncSystem := "HeatingPLC_vAI_Vars".vAI1.iFuncSystemID,
            iFuncVar := "HeatingPLC_vAI_Vars".vAI1.iFuncVar);
END_REGION

REGION Network 2
   RUNG wire#powerrail
      "vAIadv"(rInput := "HeatingPLC_vAI_Vars".vAI2.rRawValue, rFilterValue := "HeatingPLC_vAI_Vars".vAI2.rFilterSet, rMin := "HeatingPLC_vAI_Vars".vAI2.rMin, rMax := "HeatingPLC_vAI_Vars".vAI2.rMax, rCalibration := "HeatingPLC_vAI_Vars".vAI2.rCalibration, rOutput => "HeatingPLC_vAI_Vars".vAI2.rValue)
   END_RUNG
   RUNG wire#powerrail
      "AIvars"(rInput := "HeatingPLC_vAI_Vars".vAI2.rValue, iFuncSystem := "HeatingPLC_vAI_Vars".vAI2.iFuncSystemID, iFuncVar := "HeatingPLC_vAI_Vars".vAI2.iFuncVar)
   END_RUNG
   // the same network as SCL:
   "vAIadv"(rInput := "HeatingPLC_vAI_Vars".vAI2.rRawValue,
            rFilterValue := "HeatingPLC_vAI_Vars".vAI2.rFilterSet,
            rMin := "HeatingPLC_vAI_Vars".vAI2.rMin,
            rMax := "HeatingPLC_vAI_Vars".vAI2.rMax,
            rCalibration := "HeatingPLC_vAI_Vars".vAI2.rCalibration,
            rOutput => "HeatingPLC_vAI_Vars".vAI2.rValue);
   "AIvars"(rInput := "HeatingPLC_vAI_Vars".vAI2.rValue,
            iFuncSystem := "HeatingPLC_vAI_Vars".vAI2.iFuncSystemID,
            iFuncVar := "HeatingPLC_vAI_Vars".vAI2.iFuncVar);
END_REGION

REGION Network 3
   RUNG wire#powerrail
      "vAIadv"(rInput := "HeatingPLC_vAI_Vars".vAI3.rRawValue, rFilterValue := "HeatingPLC_vAI_Vars".vAI3.rFilterSet, rMin := "HeatingPLC_vAI_Vars".vAI3.rMin, rMax := "HeatingPLC_vAI_Vars".vAI3.rMax, rCalibration := "HeatingPLC_vAI_Vars".vAI3.rCalibration, rOutput => "HeatingPLC_vAI_Vars".vAI3.rValue)
   END_RUNG
   RUNG wire#powerrail
      "AIvars"(rInput := "HeatingPLC_vAI_Vars".vAI3.rValue, iFuncSystem := "HeatingPLC_vAI_Vars".vAI3.iFuncSystemID, iFuncVar := "HeatingPLC_vAI_Vars".vAI3.iFuncVar)
   END_RUNG
   // the same network as SCL:
   "vAIadv"(rInput := "HeatingPLC_vAI_Vars".vAI3.rRawValue,
            rFilterValue := "HeatingPLC_vAI_Vars".vAI3.rFilterSet,
            rMin := "HeatingPLC_vAI_Vars".vAI3.rMin,
            rMax := "HeatingPLC_vAI_Vars".vAI3.rMax,
            rCalibration := "HeatingPLC_vAI_Vars".vAI3.rCalibration,
            rOutput => "HeatingPLC_vAI_Vars".vAI3.rValue);
   "AIvars"(rInput := "HeatingPLC_vAI_Vars".vAI3.rValue,
            iFuncSystem := "HeatingPLC_vAI_Vars".vAI3.iFuncSystemID,
            iFuncVar := "HeatingPLC_vAI_Vars".vAI3.iFuncVar);
END_REGION

REGION Network 4
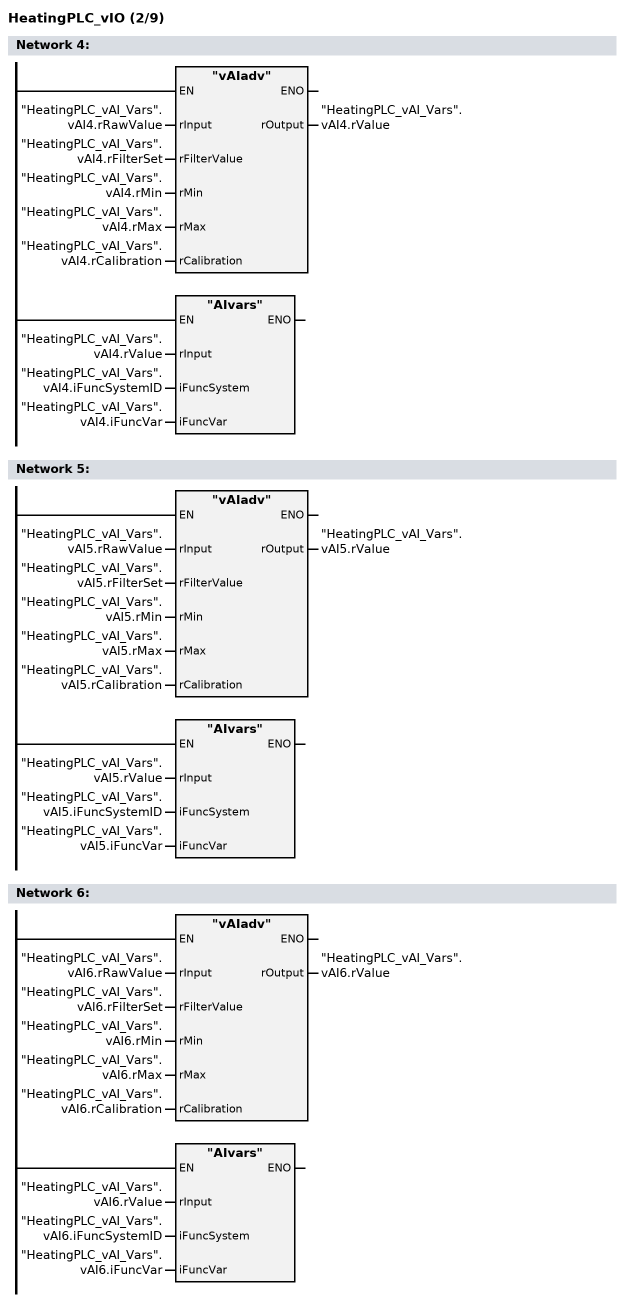
   RUNG wire#powerrail
      "vAIadv"(rInput := "HeatingPLC_vAI_Vars".vAI4.rRawValue, rFilterValue := "HeatingPLC_vAI_Vars".vAI4.rFilterSet, rMin := "HeatingPLC_vAI_Vars".vAI4.rMin, rMax := "HeatingPLC_vAI_Vars".vAI4.rMax, rCalibration := "HeatingPLC_vAI_Vars".vAI4.rCalibration, rOutput => "HeatingPLC_vAI_Vars".vAI4.rValue)
   END_RUNG
   RUNG wire#powerrail
      "AIvars"(rInput := "HeatingPLC_vAI_Vars".vAI4.rValue, iFuncSystem := "HeatingPLC_vAI_Vars".vAI4.iFuncSystemID, iFuncVar := "HeatingPLC_vAI_Vars".vAI4.iFuncVar)
   END_RUNG
   // the same network as SCL:
   "vAIadv"(rInput := "HeatingPLC_vAI_Vars".vAI4.rRawValue,
            rFilterValue := "HeatingPLC_vAI_Vars".vAI4.rFilterSet,
            rMin := "HeatingPLC_vAI_Vars".vAI4.rMin,
            rMax := "HeatingPLC_vAI_Vars".vAI4.rMax,
            rCalibration := "HeatingPLC_vAI_Vars".vAI4.rCalibration,
            rOutput => "HeatingPLC_vAI_Vars".vAI4.rValue);
   "AIvars"(rInput := "HeatingPLC_vAI_Vars".vAI4.rValue,
            iFuncSystem := "HeatingPLC_vAI_Vars".vAI4.iFuncSystemID,
            iFuncVar := "HeatingPLC_vAI_Vars".vAI4.iFuncVar);
END_REGION

REGION Network 5
   RUNG wire#powerrail
      "vAIadv"(rInput := "HeatingPLC_vAI_Vars".vAI5.rRawValue, rFilterValue := "HeatingPLC_vAI_Vars".vAI5.rFilterSet, rMin := "HeatingPLC_vAI_Vars".vAI5.rMin, rMax := "HeatingPLC_vAI_Vars".vAI5.rMax, rCalibration := "HeatingPLC_vAI_Vars".vAI5.rCalibration, rOutput => "HeatingPLC_vAI_Vars".vAI5.rValue)
   END_RUNG
   RUNG wire#powerrail
      "AIvars"(rInput := "HeatingPLC_vAI_Vars".vAI5.rValue, iFuncSystem := "HeatingPLC_vAI_Vars".vAI5.iFuncSystemID, iFuncVar := "HeatingPLC_vAI_Vars".vAI5.iFuncVar)
   END_RUNG
   // the same network as SCL:
   "vAIadv"(rInput := "HeatingPLC_vAI_Vars".vAI5.rRawValue,
            rFilterValue := "HeatingPLC_vAI_Vars".vAI5.rFilterSet,
            rMin := "HeatingPLC_vAI_Vars".vAI5.rMin,
            rMax := "HeatingPLC_vAI_Vars".vAI5.rMax,
            rCalibration := "HeatingPLC_vAI_Vars".vAI5.rCalibration,
            rOutput => "HeatingPLC_vAI_Vars".vAI5.rValue);
   "AIvars"(rInput := "HeatingPLC_vAI_Vars".vAI5.rValue,
            iFuncSystem := "HeatingPLC_vAI_Vars".vAI5.iFuncSystemID,
            iFuncVar := "HeatingPLC_vAI_Vars".vAI5.iFuncVar);
END_REGION

REGION Network 6
   RUNG wire#powerrail
      "vAIadv"(rInput := "HeatingPLC_vAI_Vars".vAI6.rRawValue, rFilterValue := "HeatingPLC_vAI_Vars".vAI6.rFilterSet, rMin := "HeatingPLC_vAI_Vars".vAI6.rMin, rMax := "HeatingPLC_vAI_Vars".vAI6.rMax, rCalibration := "HeatingPLC_vAI_Vars".vAI6.rCalibration, rOutput => "HeatingPLC_vAI_Vars".vAI6.rValue)
   END_RUNG
   RUNG wire#powerrail
      "AIvars"(rInput := "HeatingPLC_vAI_Vars".vAI6.rValue, iFuncSystem := "HeatingPLC_vAI_Vars".vAI6.iFuncSystemID, iFuncVar := "HeatingPLC_vAI_Vars".vAI6.iFuncVar)
   END_RUNG
   // the same network as SCL:
   "vAIadv"(rInput := "HeatingPLC_vAI_Vars".vAI6.rRawValue,
            rFilterValue := "HeatingPLC_vAI_Vars".vAI6.rFilterSet,
            rMin := "HeatingPLC_vAI_Vars".vAI6.rMin,
            rMax := "HeatingPLC_vAI_Vars".vAI6.rMax,
            rCalibration := "HeatingPLC_vAI_Vars".vAI6.rCalibration,
            rOutput => "HeatingPLC_vAI_Vars".vAI6.rValue);
   "AIvars"(rInput := "HeatingPLC_vAI_Vars".vAI6.rValue,
            iFuncSystem := "HeatingPLC_vAI_Vars".vAI6.iFuncSystemID,
            iFuncVar := "HeatingPLC_vAI_Vars".vAI6.iFuncVar);
END_REGION

REGION Network 7
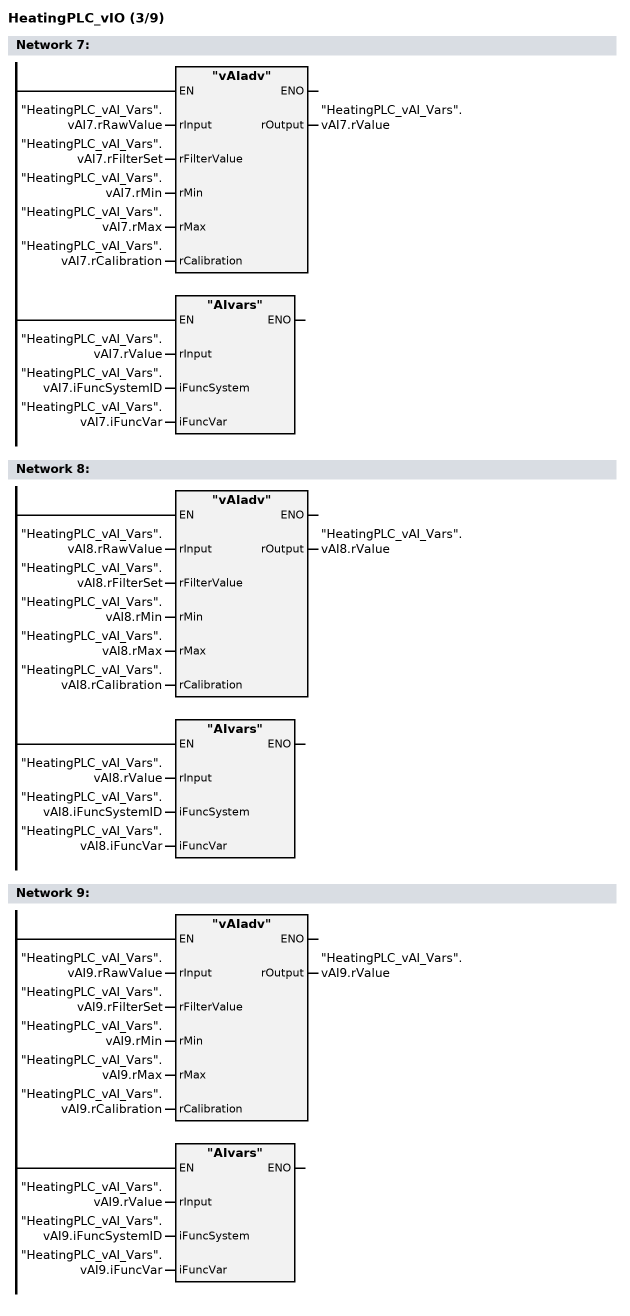
   RUNG wire#powerrail
      "vAIadv"(rInput := "HeatingPLC_vAI_Vars".vAI7.rRawValue, rFilterValue := "HeatingPLC_vAI_Vars".vAI7.rFilterSet, rMin := "HeatingPLC_vAI_Vars".vAI7.rMin, rMax := "HeatingPLC_vAI_Vars".vAI7.rMax, rCalibration := "HeatingPLC_vAI_Vars".vAI7.rCalibration, rOutput => "HeatingPLC_vAI_Vars".vAI7.rValue)
   END_RUNG
   RUNG wire#powerrail
      "AIvars"(rInput := "HeatingPLC_vAI_Vars".vAI7.rValue, iFuncSystem := "HeatingPLC_vAI_Vars".vAI7.iFuncSystemID, iFuncVar := "HeatingPLC_vAI_Vars".vAI7.iFuncVar)
   END_RUNG
   // the same network as SCL:
   "vAIadv"(rInput := "HeatingPLC_vAI_Vars".vAI7.rRawValue,
            rFilterValue := "HeatingPLC_vAI_Vars".vAI7.rFilterSet,
            rMin := "HeatingPLC_vAI_Vars".vAI7.rMin,
            rMax := "HeatingPLC_vAI_Vars".vAI7.rMax,
            rCalibration := "HeatingPLC_vAI_Vars".vAI7.rCalibration,
            rOutput => "HeatingPLC_vAI_Vars".vAI7.rValue);
   "AIvars"(rInput := "HeatingPLC_vAI_Vars".vAI7.rValue,
            iFuncSystem := "HeatingPLC_vAI_Vars".vAI7.iFuncSystemID,
            iFuncVar := "HeatingPLC_vAI_Vars".vAI7.iFuncVar);
END_REGION

REGION Network 8
   RUNG wire#powerrail
      "vAIadv"(rInput := "HeatingPLC_vAI_Vars".vAI8.rRawValue, rFilterValue := "HeatingPLC_vAI_Vars".vAI8.rFilterSet, rMin := "HeatingPLC_vAI_Vars".vAI8.rMin, rMax := "HeatingPLC_vAI_Vars".vAI8.rMax, rCalibration := "HeatingPLC_vAI_Vars".vAI8.rCalibration, rOutput => "HeatingPLC_vAI_Vars".vAI8.rValue)
   END_RUNG
   RUNG wire#powerrail
      "AIvars"(rInput := "HeatingPLC_vAI_Vars".vAI8.rValue, iFuncSystem := "HeatingPLC_vAI_Vars".vAI8.iFuncSystemID, iFuncVar := "HeatingPLC_vAI_Vars".vAI8.iFuncVar)
   END_RUNG
   // the same network as SCL:
   "vAIadv"(rInput := "HeatingPLC_vAI_Vars".vAI8.rRawValue,
            rFilterValue := "HeatingPLC_vAI_Vars".vAI8.rFilterSet,
            rMin := "HeatingPLC_vAI_Vars".vAI8.rMin,
            rMax := "HeatingPLC_vAI_Vars".vAI8.rMax,
            rCalibration := "HeatingPLC_vAI_Vars".vAI8.rCalibration,
            rOutput => "HeatingPLC_vAI_Vars".vAI8.rValue);
   "AIvars"(rInput := "HeatingPLC_vAI_Vars".vAI8.rValue,
            iFuncSystem := "HeatingPLC_vAI_Vars".vAI8.iFuncSystemID,
            iFuncVar := "HeatingPLC_vAI_Vars".vAI8.iFuncVar);
END_REGION

REGION Network 9
   RUNG wire#powerrail
      "vAIadv"(rInput := "HeatingPLC_vAI_Vars".vAI9.rRawValue, rFilterValue := "HeatingPLC_vAI_Vars".vAI9.rFilterSet, rMin := "HeatingPLC_vAI_Vars".vAI9.rMin, rMax := "HeatingPLC_vAI_Vars".vAI9.rMax, rCalibration := "HeatingPLC_vAI_Vars".vAI9.rCalibration, rOutput => "HeatingPLC_vAI_Vars".vAI9.rValue)
   END_RUNG
   RUNG wire#powerrail
      "AIvars"(rInput := "HeatingPLC_vAI_Vars".vAI9.rValue, iFuncSystem := "HeatingPLC_vAI_Vars".vAI9.iFuncSystemID, iFuncVar := "HeatingPLC_vAI_Vars".vAI9.iFuncVar)
   END_RUNG
   // the same network as SCL:
   "vAIadv"(rInput := "HeatingPLC_vAI_Vars".vAI9.rRawValue,
            rFilterValue := "HeatingPLC_vAI_Vars".vAI9.rFilterSet,
            rMin := "HeatingPLC_vAI_Vars".vAI9.rMin,
            rMax := "HeatingPLC_vAI_Vars".vAI9.rMax,
            rCalibration := "HeatingPLC_vAI_Vars".vAI9.rCalibration,
            rOutput => "HeatingPLC_vAI_Vars".vAI9.rValue);
   "AIvars"(rInput := "HeatingPLC_vAI_Vars".vAI9.rValue,
            iFuncSystem := "HeatingPLC_vAI_Vars".vAI9.iFuncSystemID,
            iFuncVar := "HeatingPLC_vAI_Vars".vAI9.iFuncVar);
END_REGION

REGION Network 10
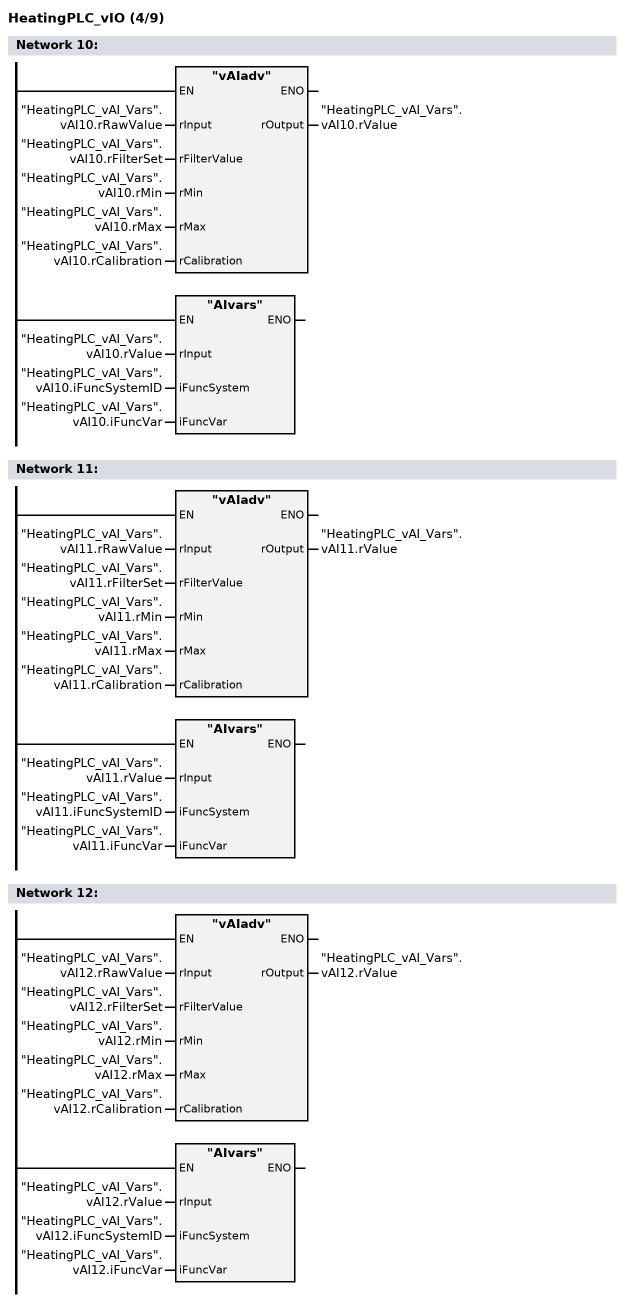
   RUNG wire#powerrail
      "vAIadv"(rInput := "HeatingPLC_vAI_Vars".vAI10.rRawValue, rFilterValue := "HeatingPLC_vAI_Vars".vAI10.rFilterSet, rMin := "HeatingPLC_vAI_Vars".vAI10.rMin, rMax := "HeatingPLC_vAI_Vars".vAI10.rMax, rCalibration := "HeatingPLC_vAI_Vars".vAI10.rCalibration, rOutput => "HeatingPLC_vAI_Vars".vAI10.rValue)
   END_RUNG
   RUNG wire#powerrail
      "AIvars"(rInput := "HeatingPLC_vAI_Vars".vAI10.rValue, iFuncSystem := "HeatingPLC_vAI_Vars".vAI10.iFuncSystemID, iFuncVar := "HeatingPLC_vAI_Vars".vAI10.iFuncVar)
   END_RUNG
   // the same network as SCL:
   "vAIadv"(rInput := "HeatingPLC_vAI_Vars".vAI10.rRawValue,
            rFilterValue := "HeatingPLC_vAI_Vars".vAI10.rFilterSet,
            rMin := "HeatingPLC_vAI_Vars".vAI10.rMin,
            rMax := "HeatingPLC_vAI_Vars".vAI10.rMax,
            rCalibration := "HeatingPLC_vAI_Vars".vAI10.rCalibration,
            rOutput => "HeatingPLC_vAI_Vars".vAI10.rValue);
   "AIvars"(rInput := "HeatingPLC_vAI_Vars".vAI10.rValue,
            iFuncSystem := "HeatingPLC_vAI_Vars".vAI10.iFuncSystemID,
            iFuncVar := "HeatingPLC_vAI_Vars".vAI10.iFuncVar);
END_REGION

REGION Network 11
   RUNG wire#powerrail
      "vAIadv"(rInput := "HeatingPLC_vAI_Vars".vAI11.rRawValue, rFilterValue := "HeatingPLC_vAI_Vars".vAI11.rFilterSet, rMin := "HeatingPLC_vAI_Vars".vAI11.rMin, rMax := "HeatingPLC_vAI_Vars".vAI11.rMax, rCalibration := "HeatingPLC_vAI_Vars".vAI11.rCalibration, rOutput => "HeatingPLC_vAI_Vars".vAI11.rValue)
   END_RUNG
   RUNG wire#powerrail
      "AIvars"(rInput := "HeatingPLC_vAI_Vars".vAI11.rValue, iFuncSystem := "HeatingPLC_vAI_Vars".vAI11.iFuncSystemID, iFuncVar := "HeatingPLC_vAI_Vars".vAI11.iFuncVar)
   END_RUNG
   // the same network as SCL:
   "vAIadv"(rInput := "HeatingPLC_vAI_Vars".vAI11.rRawValue,
            rFilterValue := "HeatingPLC_vAI_Vars".vAI11.rFilterSet,
            rMin := "HeatingPLC_vAI_Vars".vAI11.rMin,
            rMax := "HeatingPLC_vAI_Vars".vAI11.rMax,
            rCalibration := "HeatingPLC_vAI_Vars".vAI11.rCalibration,
            rOutput => "HeatingPLC_vAI_Vars".vAI11.rValue);
   "AIvars"(rInput := "HeatingPLC_vAI_Vars".vAI11.rValue,
            iFuncSystem := "HeatingPLC_vAI_Vars".vAI11.iFuncSystemID,
            iFuncVar := "HeatingPLC_vAI_Vars".vAI11.iFuncVar);
END_REGION

REGION Network 12
   RUNG wire#powerrail
      "vAIadv"(rInput := "HeatingPLC_vAI_Vars".vAI12.rRawValue, rFilterValue := "HeatingPLC_vAI_Vars".vAI12.rFilterSet, rMin := "HeatingPLC_vAI_Vars".vAI12.rMin, rMax := "HeatingPLC_vAI_Vars".vAI12.rMax, rCalibration := "HeatingPLC_vAI_Vars".vAI12.rCalibration, rOutput => "HeatingPLC_vAI_Vars".vAI12.rValue)
   END_RUNG
   RUNG wire#powerrail
      "AIvars"(rInput := "HeatingPLC_vAI_Vars".vAI12.rValue, iFuncSystem := "HeatingPLC_vAI_Vars".vAI12.iFuncSystemID, iFuncVar := "HeatingPLC_vAI_Vars".vAI12.iFuncVar)
   END_RUNG
   // the same network as SCL:
   "vAIadv"(rInput := "HeatingPLC_vAI_Vars".vAI12.rRawValue,
            rFilterValue := "HeatingPLC_vAI_Vars".vAI12.rFilterSet,
            rMin := "HeatingPLC_vAI_Vars".vAI12.rMin,
            rMax := "HeatingPLC_vAI_Vars".vAI12.rMax,
            rCalibration := "HeatingPLC_vAI_Vars".vAI12.rCalibration,
            rOutput => "HeatingPLC_vAI_Vars".vAI12.rValue);
   "AIvars"(rInput := "HeatingPLC_vAI_Vars".vAI12.rValue,
            iFuncSystem := "HeatingPLC_vAI_Vars".vAI12.iFuncSystemID,
            iFuncVar := "HeatingPLC_vAI_Vars".vAI12.iFuncVar);
END_REGION

REGION Network 13
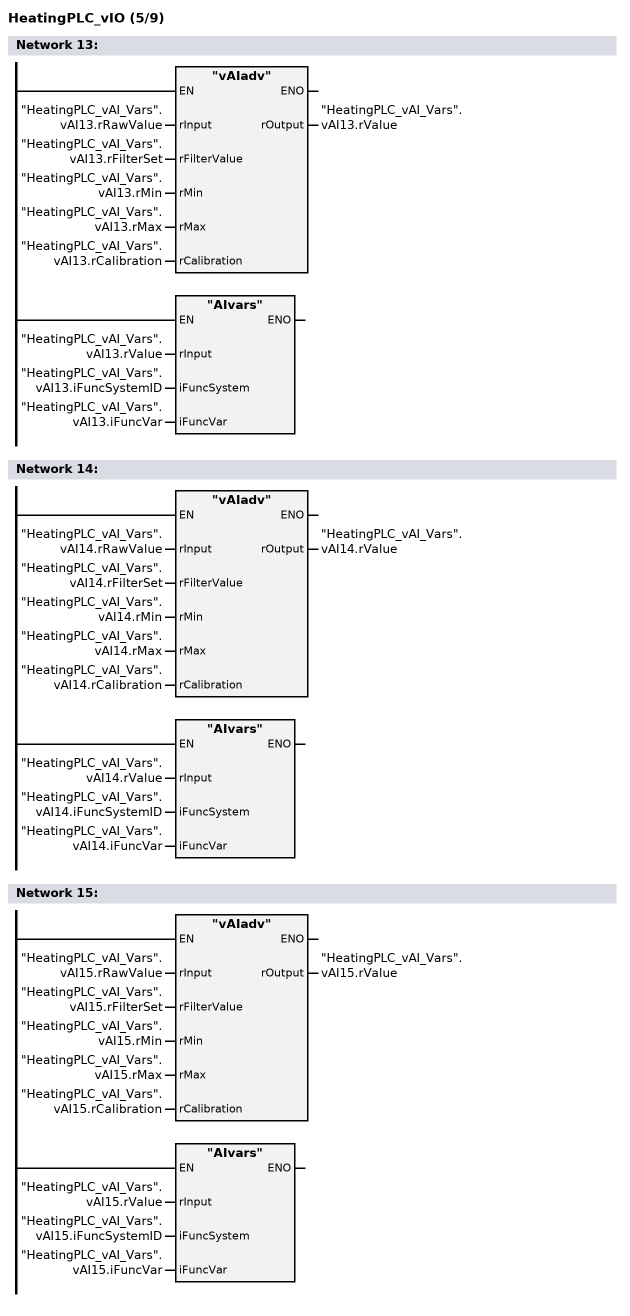
   RUNG wire#powerrail
      "vAIadv"(rInput := "HeatingPLC_vAI_Vars".vAI13.rRawValue, rFilterValue := "HeatingPLC_vAI_Vars".vAI13.rFilterSet, rMin := "HeatingPLC_vAI_Vars".vAI13.rMin, rMax := "HeatingPLC_vAI_Vars".vAI13.rMax, rCalibration := "HeatingPLC_vAI_Vars".vAI13.rCalibration, rOutput => "HeatingPLC_vAI_Vars".vAI13.rValue)
   END_RUNG
   RUNG wire#powerrail
      "AIvars"(rInput := "HeatingPLC_vAI_Vars".vAI13.rValue, iFuncSystem := "HeatingPLC_vAI_Vars".vAI13.iFuncSystemID, iFuncVar := "HeatingPLC_vAI_Vars".vAI13.iFuncVar)
   END_RUNG
   // the same network as SCL:
   "vAIadv"(rInput := "HeatingPLC_vAI_Vars".vAI13.rRawValue,
            rFilterValue := "HeatingPLC_vAI_Vars".vAI13.rFilterSet,
            rMin := "HeatingPLC_vAI_Vars".vAI13.rMin,
            rMax := "HeatingPLC_vAI_Vars".vAI13.rMax,
            rCalibration := "HeatingPLC_vAI_Vars".vAI13.rCalibration,
            rOutput => "HeatingPLC_vAI_Vars".vAI13.rValue);
   "AIvars"(rInput := "HeatingPLC_vAI_Vars".vAI13.rValue,
            iFuncSystem := "HeatingPLC_vAI_Vars".vAI13.iFuncSystemID,
            iFuncVar := "HeatingPLC_vAI_Vars".vAI13.iFuncVar);
END_REGION

REGION Network 14
   RUNG wire#powerrail
      "vAIadv"(rInput := "HeatingPLC_vAI_Vars".vAI14.rRawValue, rFilterValue := "HeatingPLC_vAI_Vars".vAI14.rFilterSet, rMin := "HeatingPLC_vAI_Vars".vAI14.rMin, rMax := "HeatingPLC_vAI_Vars".vAI14.rMax, rCalibration := "HeatingPLC_vAI_Vars".vAI14.rCalibration, rOutput => "HeatingPLC_vAI_Vars".vAI14.rValue)
   END_RUNG
   RUNG wire#powerrail
      "AIvars"(rInput := "HeatingPLC_vAI_Vars".vAI14.rValue, iFuncSystem := "HeatingPLC_vAI_Vars".vAI14.iFuncSystemID, iFuncVar := "HeatingPLC_vAI_Vars".vAI14.iFuncVar)
   END_RUNG
   // the same network as SCL:
   "vAIadv"(rInput := "HeatingPLC_vAI_Vars".vAI14.rRawValue,
            rFilterValue := "HeatingPLC_vAI_Vars".vAI14.rFilterSet,
            rMin := "HeatingPLC_vAI_Vars".vAI14.rMin,
            rMax := "HeatingPLC_vAI_Vars".vAI14.rMax,
            rCalibration := "HeatingPLC_vAI_Vars".vAI14.rCalibration,
            rOutput => "HeatingPLC_vAI_Vars".vAI14.rValue);
   "AIvars"(rInput := "HeatingPLC_vAI_Vars".vAI14.rValue,
            iFuncSystem := "HeatingPLC_vAI_Vars".vAI14.iFuncSystemID,
            iFuncVar := "HeatingPLC_vAI_Vars".vAI14.iFuncVar);
END_REGION

REGION Network 15
   RUNG wire#powerrail
      "vAIadv"(rInput := "HeatingPLC_vAI_Vars".vAI15.rRawValue, rFilterValue := "HeatingPLC_vAI_Vars".vAI15.rFilterSet, rMin := "HeatingPLC_vAI_Vars".vAI15.rMin, rMax := "HeatingPLC_vAI_Vars".vAI15.rMax, rCalibration := "HeatingPLC_vAI_Vars".vAI15.rCalibration, rOutput => "HeatingPLC_vAI_Vars".vAI15.rValue)
   END_RUNG
   RUNG wire#powerrail
      "AIvars"(rInput := "HeatingPLC_vAI_Vars".vAI15.rValue, iFuncSystem := "HeatingPLC_vAI_Vars".vAI15.iFuncSystemID, iFuncVar := "HeatingPLC_vAI_Vars".vAI15.iFuncVar)
   END_RUNG
   // the same network as SCL:
   "vAIadv"(rInput := "HeatingPLC_vAI_Vars".vAI15.rRawValue,
            rFilterValue := "HeatingPLC_vAI_Vars".vAI15.rFilterSet,
            rMin := "HeatingPLC_vAI_Vars".vAI15.rMin,
            rMax := "HeatingPLC_vAI_Vars".vAI15.rMax,
            rCalibration := "HeatingPLC_vAI_Vars".vAI15.rCalibration,
            rOutput => "HeatingPLC_vAI_Vars".vAI15.rValue);
   "AIvars"(rInput := "HeatingPLC_vAI_Vars".vAI15.rValue,
            iFuncSystem := "HeatingPLC_vAI_Vars".vAI15.iFuncSystemID,
            iFuncVar := "HeatingPLC_vAI_Vars".vAI15.iFuncVar);
END_REGION

REGION Network 16
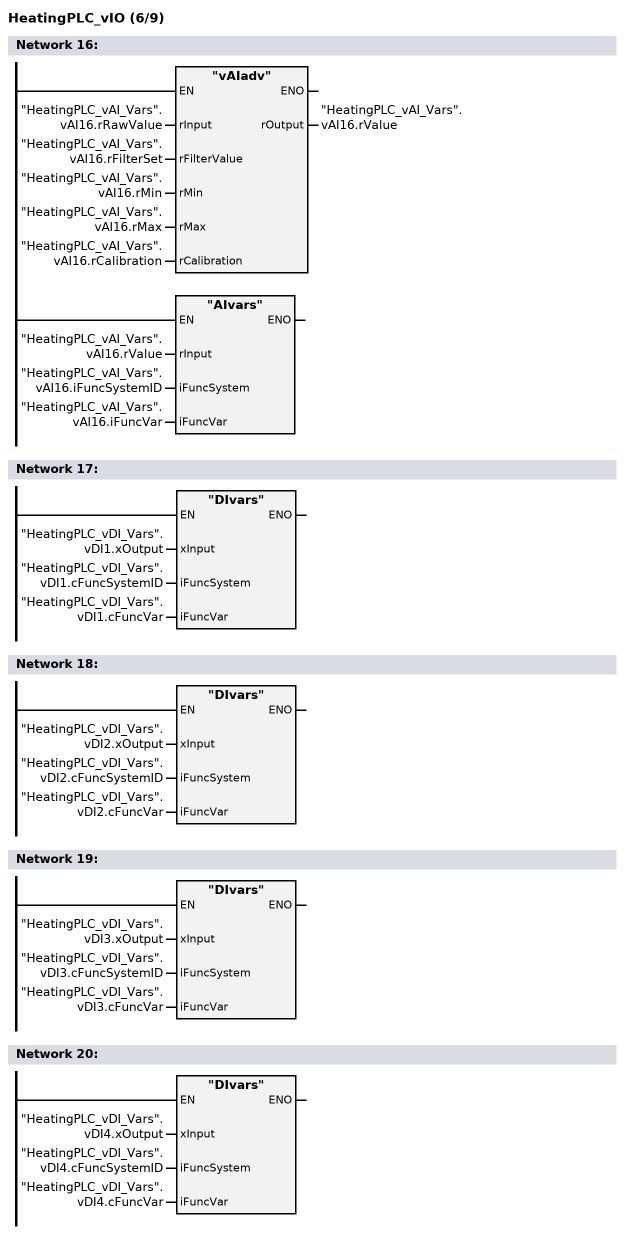
   RUNG wire#powerrail
      "vAIadv"(rInput := "HeatingPLC_vAI_Vars".vAI16.rRawValue, rFilterValue := "HeatingPLC_vAI_Vars".vAI16.rFilterSet, rMin := "HeatingPLC_vAI_Vars".vAI16.rMin, rMax := "HeatingPLC_vAI_Vars".vAI16.rMax, rCalibration := "HeatingPLC_vAI_Vars".vAI16.rCalibration, rOutput => "HeatingPLC_vAI_Vars".vAI16.rValue)
   END_RUNG
   RUNG wire#powerrail
      "AIvars"(rInput := "HeatingPLC_vAI_Vars".vAI16.rValue, iFuncSystem := "HeatingPLC_vAI_Vars".vAI16.iFuncSystemID, iFuncVar := "HeatingPLC_vAI_Vars".vAI16.iFuncVar)
   END_RUNG
   // the same network as SCL:
   "vAIadv"(rInput := "HeatingPLC_vAI_Vars".vAI16.rRawValue,
            rFilterValue := "HeatingPLC_vAI_Vars".vAI16.rFilterSet,
            rMin := "HeatingPLC_vAI_Vars".vAI16.rMin,
            rMax := "HeatingPLC_vAI_Vars".vAI16.rMax,
            rCalibration := "HeatingPLC_vAI_Vars".vAI16.rCalibration,
            rOutput => "HeatingPLC_vAI_Vars".vAI16.rValue);
   "AIvars"(rInput := "HeatingPLC_vAI_Vars".vAI16.rValue,
            iFuncSystem := "HeatingPLC_vAI_Vars".vAI16.iFuncSystemID,
            iFuncVar := "HeatingPLC_vAI_Vars".vAI16.iFuncVar);
END_REGION

REGION Network 17
   RUNG wire#powerrail
      "DIvars"(xInput := "HeatingPLC_vDI_Vars".vDI1.xOutput, iFuncSystem := "HeatingPLC_vDI_Vars".vDI1.cFuncSystemID, iFuncVar := "HeatingPLC_vDI_Vars".vDI1.cFuncVar)
   END_RUNG
   // the same network as SCL:
   "DIvars"(xInput := "HeatingPLC_vDI_Vars".vDI1.xOutput,
            iFuncSystem := "HeatingPLC_vDI_Vars".vDI1.cFuncSystemID,
            iFuncVar := "HeatingPLC_vDI_Vars".vDI1.cFuncVar);
END_REGION

REGION Network 18
   RUNG wire#powerrail
      "DIvars"(xInput := "HeatingPLC_vDI_Vars".vDI2.xOutput, iFuncSystem := "HeatingPLC_vDI_Vars".vDI2.cFuncSystemID, iFuncVar := "HeatingPLC_vDI_Vars".vDI2.cFuncVar)
   END_RUNG
   // the same network as SCL:
   "DIvars"(xInput := "HeatingPLC_vDI_Vars".vDI2.xOutput,
            iFuncSystem := "HeatingPLC_vDI_Vars".vDI2.cFuncSystemID,
            iFuncVar := "HeatingPLC_vDI_Vars".vDI2.cFuncVar);
END_REGION

REGION Network 19
   RUNG wire#powerrail
      "DIvars"(xInput := "HeatingPLC_vDI_Vars".vDI3.xOutput, iFuncSystem := "HeatingPLC_vDI_Vars".vDI3.cFuncSystemID, iFuncVar := "HeatingPLC_vDI_Vars".vDI3.cFuncVar)
   END_RUNG
   // the same network as SCL:
   "DIvars"(xInput := "HeatingPLC_vDI_Vars".vDI3.xOutput,
            iFuncSystem := "HeatingPLC_vDI_Vars".vDI3.cFuncSystemID,
            iFuncVar := "HeatingPLC_vDI_Vars".vDI3.cFuncVar);
END_REGION

REGION Network 20
   RUNG wire#powerrail
      "DIvars"(xInput := "HeatingPLC_vDI_Vars".vDI4.xOutput, iFuncSystem := "HeatingPLC_vDI_Vars".vDI4.cFuncSystemID, iFuncVar := "HeatingPLC_vDI_Vars".vDI4.cFuncVar)
   END_RUNG
   // the same network as SCL:
   "DIvars"(xInput := "HeatingPLC_vDI_Vars".vDI4.xOutput,
            iFuncSystem := "HeatingPLC_vDI_Vars".vDI4.cFuncSystemID,
            iFuncVar := "HeatingPLC_vDI_Vars".vDI4.cFuncVar);
END_REGION

REGION Network 21
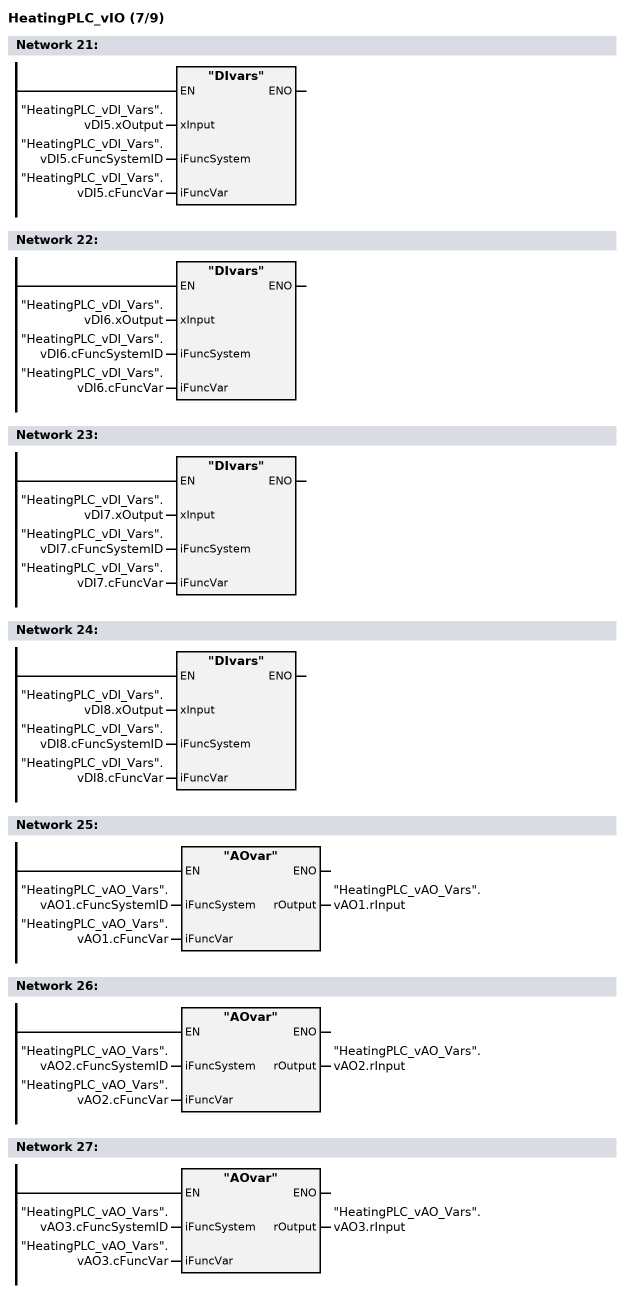
   RUNG wire#powerrail
      "DIvars"(xInput := "HeatingPLC_vDI_Vars".vDI5.xOutput, iFuncSystem := "HeatingPLC_vDI_Vars".vDI5.cFuncSystemID, iFuncVar := "HeatingPLC_vDI_Vars".vDI5.cFuncVar)
   END_RUNG
   // the same network as SCL:
   "DIvars"(xInput := "HeatingPLC_vDI_Vars".vDI5.xOutput,
            iFuncSystem := "HeatingPLC_vDI_Vars".vDI5.cFuncSystemID,
            iFuncVar := "HeatingPLC_vDI_Vars".vDI5.cFuncVar);
END_REGION

REGION Network 22
   RUNG wire#powerrail
      "DIvars"(xInput := "HeatingPLC_vDI_Vars".vDI6.xOutput, iFuncSystem := "HeatingPLC_vDI_Vars".vDI6.cFuncSystemID, iFuncVar := "HeatingPLC_vDI_Vars".vDI6.cFuncVar)
   END_RUNG
   // the same network as SCL:
   "DIvars"(xInput := "HeatingPLC_vDI_Vars".vDI6.xOutput,
            iFuncSystem := "HeatingPLC_vDI_Vars".vDI6.cFuncSystemID,
            iFuncVar := "HeatingPLC_vDI_Vars".vDI6.cFuncVar);
END_REGION

REGION Network 23
   RUNG wire#powerrail
      "DIvars"(xInput := "HeatingPLC_vDI_Vars".vDI7.xOutput, iFuncSystem := "HeatingPLC_vDI_Vars".vDI7.cFuncSystemID, iFuncVar := "HeatingPLC_vDI_Vars".vDI7.cFuncVar)
   END_RUNG
   // the same network as SCL:
   "DIvars"(xInput := "HeatingPLC_vDI_Vars".vDI7.xOutput,
            iFuncSystem := "HeatingPLC_vDI_Vars".vDI7.cFuncSystemID,
            iFuncVar := "HeatingPLC_vDI_Vars".vDI7.cFuncVar);
END_REGION

REGION Network 24
   RUNG wire#powerrail
      "DIvars"(xInput := "HeatingPLC_vDI_Vars".vDI8.xOutput, iFuncSystem := "HeatingPLC_vDI_Vars".vDI8.cFuncSystemID, iFuncVar := "HeatingPLC_vDI_Vars".vDI8.cFuncVar)
   END_RUNG
   // the same network as SCL:
   "DIvars"(xInput := "HeatingPLC_vDI_Vars".vDI8.xOutput,
            iFuncSystem := "HeatingPLC_vDI_Vars".vDI8.cFuncSystemID,
            iFuncVar := "HeatingPLC_vDI_Vars".vDI8.cFuncVar);
END_REGION

REGION Network 25
   RUNG wire#powerrail
      "AOvar"(iFuncSystem := "HeatingPLC_vAO_Vars".vAO1.cFuncSystemID, iFuncVar := "HeatingPLC_vAO_Vars".vAO1.cFuncVar, rOutput => "HeatingPLC_vAO_Vars".vAO1.rInput)
   END_RUNG
   // the same network as SCL:
   "AOvar"(iFuncSystem := "HeatingPLC_vAO_Vars".vAO1.cFuncSystemID,
           iFuncVar := "HeatingPLC_vAO_Vars".vAO1.cFuncVar,
           rOutput => "HeatingPLC_vAO_Vars".vAO1.rInput);
END_REGION

REGION Network 26
   RUNG wire#powerrail
      "AOvar"(iFuncSystem := "HeatingPLC_vAO_Vars".vAO2.cFuncSystemID, iFuncVar := "HeatingPLC_vAO_Vars".vAO2.cFuncVar, rOutput => "HeatingPLC_vAO_Vars".vAO2.rInput)
   END_RUNG
   // the same network as SCL:
   "AOvar"(iFuncSystem := "HeatingPLC_vAO_Vars".vAO2.cFuncSystemID,
           iFuncVar := "HeatingPLC_vAO_Vars".vAO2.cFuncVar,
           rOutput => "HeatingPLC_vAO_Vars".vAO2.rInput);
END_REGION

REGION Network 27
   RUNG wire#powerrail
      "AOvar"(iFuncSystem := "HeatingPLC_vAO_Vars".vAO3.cFuncSystemID, iFuncVar := "HeatingPLC_vAO_Vars".vAO3.cFuncVar, rOutput => "HeatingPLC_vAO_Vars".vAO3.rInput)
   END_RUNG
   // the same network as SCL:
   "AOvar"(iFuncSystem := "HeatingPLC_vAO_Vars".vAO3.cFuncSystemID,
           iFuncVar := "HeatingPLC_vAO_Vars".vAO3.cFuncVar,
           rOutput => "HeatingPLC_vAO_Vars".vAO3.rInput);
END_REGION

REGION Network 28
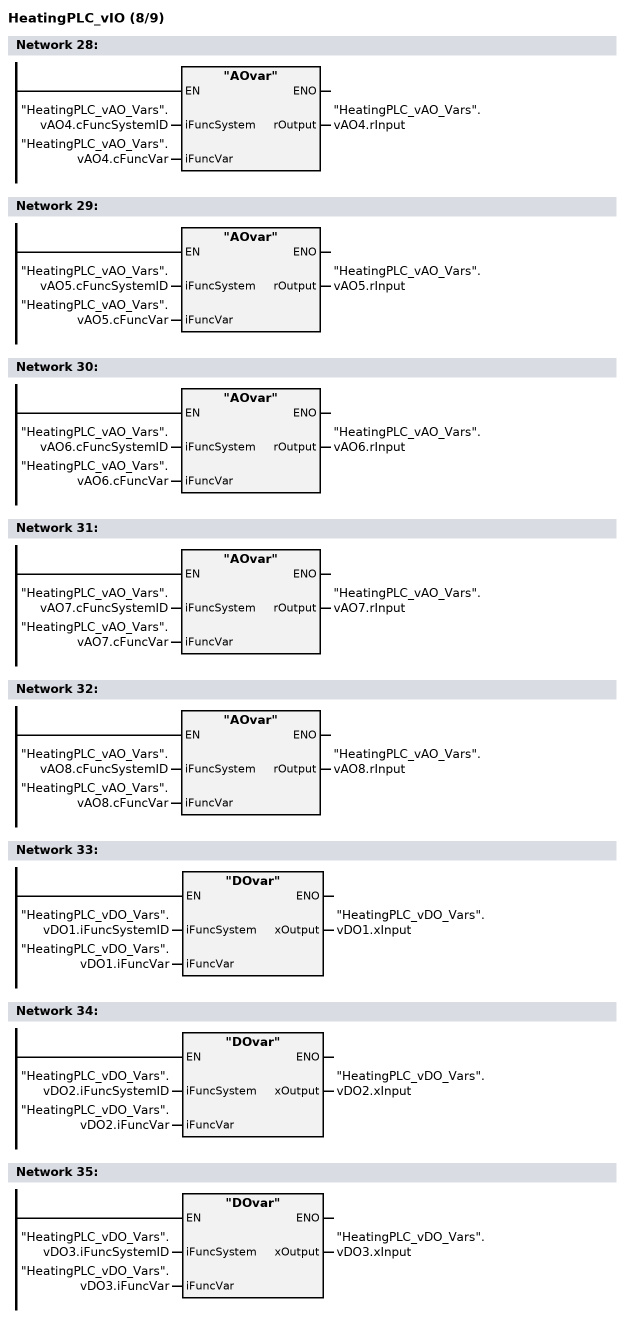
   RUNG wire#powerrail
      "AOvar"(iFuncSystem := "HeatingPLC_vAO_Vars".vAO4.cFuncSystemID, iFuncVar := "HeatingPLC_vAO_Vars".vAO4.cFuncVar, rOutput => "HeatingPLC_vAO_Vars".vAO4.rInput)
   END_RUNG
   // the same network as SCL:
   "AOvar"(iFuncSystem := "HeatingPLC_vAO_Vars".vAO4.cFuncSystemID,
           iFuncVar := "HeatingPLC_vAO_Vars".vAO4.cFuncVar,
           rOutput => "HeatingPLC_vAO_Vars".vAO4.rInput);
END_REGION

REGION Network 29
   RUNG wire#powerrail
      "AOvar"(iFuncSystem := "HeatingPLC_vAO_Vars".vAO5.cFuncSystemID, iFuncVar := "HeatingPLC_vAO_Vars".vAO5.cFuncVar, rOutput => "HeatingPLC_vAO_Vars".vAO5.rInput)
   END_RUNG
   // the same network as SCL:
   "AOvar"(iFuncSystem := "HeatingPLC_vAO_Vars".vAO5.cFuncSystemID,
           iFuncVar := "HeatingPLC_vAO_Vars".vAO5.cFuncVar,
           rOutput => "HeatingPLC_vAO_Vars".vAO5.rInput);
END_REGION

REGION Network 30
   RUNG wire#powerrail
      "AOvar"(iFuncSystem := "HeatingPLC_vAO_Vars".vAO6.cFuncSystemID, iFuncVar := "HeatingPLC_vAO_Vars".vAO6.cFuncVar, rOutput => "HeatingPLC_vAO_Vars".vAO6.rInput)
   END_RUNG
   // the same network as SCL:
   "AOvar"(iFuncSystem := "HeatingPLC_vAO_Vars".vAO6.cFuncSystemID,
           iFuncVar := "HeatingPLC_vAO_Vars".vAO6.cFuncVar,
           rOutput => "HeatingPLC_vAO_Vars".vAO6.rInput);
END_REGION

REGION Network 31
   RUNG wire#powerrail
      "AOvar"(iFuncSystem := "HeatingPLC_vAO_Vars".vAO7.cFuncSystemID, iFuncVar := "HeatingPLC_vAO_Vars".vAO7.cFuncVar, rOutput => "HeatingPLC_vAO_Vars".vAO7.rInput)
   END_RUNG
   // the same network as SCL:
   "AOvar"(iFuncSystem := "HeatingPLC_vAO_Vars".vAO7.cFuncSystemID,
           iFuncVar := "HeatingPLC_vAO_Vars".vAO7.cFuncVar,
           rOutput => "HeatingPLC_vAO_Vars".vAO7.rInput);
END_REGION

REGION Network 32
   RUNG wire#powerrail
      "AOvar"(iFuncSystem := "HeatingPLC_vAO_Vars".vAO8.cFuncSystemID, iFuncVar := "HeatingPLC_vAO_Vars".vAO8.cFuncVar, rOutput => "HeatingPLC_vAO_Vars".vAO8.rInput)
   END_RUNG
   // the same network as SCL:
   "AOvar"(iFuncSystem := "HeatingPLC_vAO_Vars".vAO8.cFuncSystemID,
           iFuncVar := "HeatingPLC_vAO_Vars".vAO8.cFuncVar,
           rOutput => "HeatingPLC_vAO_Vars".vAO8.rInput);
END_REGION

REGION Network 33
   RUNG wire#powerrail
      "DOvar"(iFuncSystem := "HeatingPLC_vDO_Vars".vDO1.iFuncSystemID, iFuncVar := "HeatingPLC_vDO_Vars".vDO1.iFuncVar, xOutput => "HeatingPLC_vDO_Vars".vDO1.xInput)
   END_RUNG
   // the same network as SCL:
   "DOvar"(iFuncSystem := "HeatingPLC_vDO_Vars".vDO1.iFuncSystemID,
           iFuncVar := "HeatingPLC_vDO_Vars".vDO1.iFuncVar,
           xOutput => "HeatingPLC_vDO_Vars".vDO1.xInput);
END_REGION

REGION Network 34
   RUNG wire#powerrail
      "DOvar"(iFuncSystem := "HeatingPLC_vDO_Vars".vDO2.iFuncSystemID, iFuncVar := "HeatingPLC_vDO_Vars".vDO2.iFuncVar, xOutput => "HeatingPLC_vDO_Vars".vDO2.xInput)
   END_RUNG
   // the same network as SCL:
   "DOvar"(iFuncSystem := "HeatingPLC_vDO_Vars".vDO2.iFuncSystemID,
           iFuncVar := "HeatingPLC_vDO_Vars".vDO2.iFuncVar,
           xOutput => "HeatingPLC_vDO_Vars".vDO2.xInput);
END_REGION

REGION Network 35
   RUNG wire#powerrail
      "DOvar"(iFuncSystem := "HeatingPLC_vDO_Vars".vDO3.iFuncSystemID, iFuncVar := "HeatingPLC_vDO_Vars".vDO3.iFuncVar, xOutput => "HeatingPLC_vDO_Vars".vDO3.xInput)
   END_RUNG
   // the same network as SCL:
   "DOvar"(iFuncSystem := "HeatingPLC_vDO_Vars".vDO3.iFuncSystemID,
           iFuncVar := "HeatingPLC_vDO_Vars".vDO3.iFuncVar,
           xOutput => "HeatingPLC_vDO_Vars".vDO3.xInput);
END_REGION

REGION Network 36
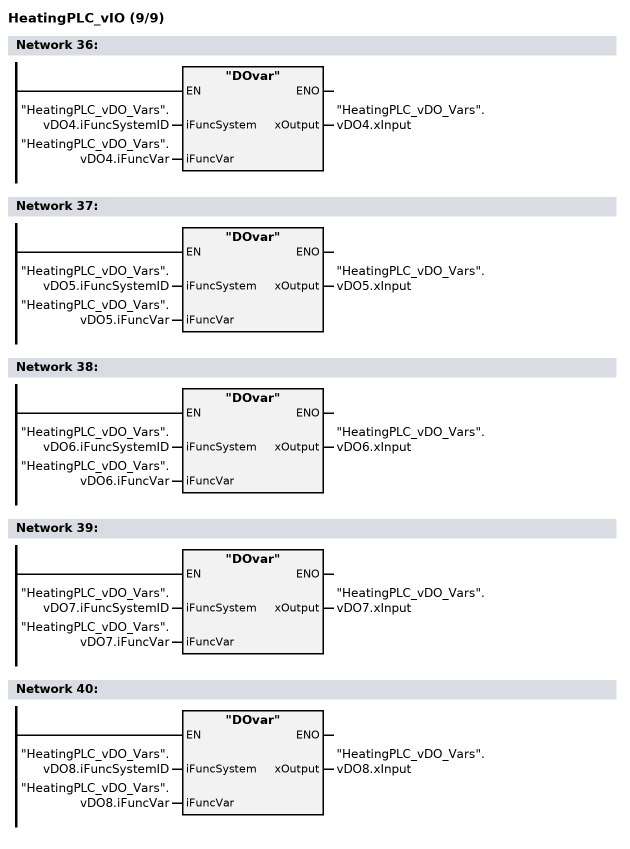
   RUNG wire#powerrail
      "DOvar"(iFuncSystem := "HeatingPLC_vDO_Vars".vDO4.iFuncSystemID, iFuncVar := "HeatingPLC_vDO_Vars".vDO4.iFuncVar, xOutput => "HeatingPLC_vDO_Vars".vDO4.xInput)
   END_RUNG
   // the same network as SCL:
   "DOvar"(iFuncSystem := "HeatingPLC_vDO_Vars".vDO4.iFuncSystemID,
           iFuncVar := "HeatingPLC_vDO_Vars".vDO4.iFuncVar,
           xOutput => "HeatingPLC_vDO_Vars".vDO4.xInput);
END_REGION

REGION Network 37
   RUNG wire#powerrail
      "DOvar"(iFuncSystem := "HeatingPLC_vDO_Vars".vDO5.iFuncSystemID, iFuncVar := "HeatingPLC_vDO_Vars".vDO5.iFuncVar, xOutput => "HeatingPLC_vDO_Vars".vDO5.xInput)
   END_RUNG
   // the same network as SCL:
   "DOvar"(iFuncSystem := "HeatingPLC_vDO_Vars".vDO5.iFuncSystemID,
           iFuncVar := "HeatingPLC_vDO_Vars".vDO5.iFuncVar,
           xOutput => "HeatingPLC_vDO_Vars".vDO5.xInput);
END_REGION

REGION Network 38
   RUNG wire#powerrail
      "DOvar"(iFuncSystem := "HeatingPLC_vDO_Vars".vDO6.iFuncSystemID, iFuncVar := "HeatingPLC_vDO_Vars".vDO6.iFuncVar, xOutput => "HeatingPLC_vDO_Vars".vDO6.xInput)
   END_RUNG
   // the same network as SCL:
   "DOvar"(iFuncSystem := "HeatingPLC_vDO_Vars".vDO6.iFuncSystemID,
           iFuncVar := "HeatingPLC_vDO_Vars".vDO6.iFuncVar,
           xOutput => "HeatingPLC_vDO_Vars".vDO6.xInput);
END_REGION

REGION Network 39
   RUNG wire#powerrail
      "DOvar"(iFuncSystem := "HeatingPLC_vDO_Vars".vDO7.iFuncSystemID, iFuncVar := "HeatingPLC_vDO_Vars".vDO7.iFuncVar, xOutput => "HeatingPLC_vDO_Vars".vDO7.xInput)
   END_RUNG
   // the same network as SCL:
   "DOvar"(iFuncSystem := "HeatingPLC_vDO_Vars".vDO7.iFuncSystemID,
           iFuncVar := "HeatingPLC_vDO_Vars".vDO7.iFuncVar,
           xOutput => "HeatingPLC_vDO_Vars".vDO7.xInput);
END_REGION

REGION Network 40
   RUNG wire#powerrail
      "DOvar"(iFuncSystem := "HeatingPLC_vDO_Vars".vDO8.iFuncSystemID, iFuncVar := "HeatingPLC_vDO_Vars".vDO8.iFuncVar, xOutput => "HeatingPLC_vDO_Vars".vDO8.xInput)
   END_RUNG
   // the same network as SCL:
   "DOvar"(iFuncSystem := "HeatingPLC_vDO_Vars".vDO8.iFuncSystemID,
           iFuncVar := "HeatingPLC_vDO_Vars".vDO8.iFuncVar,
           xOutput => "HeatingPLC_vDO_Vars".vDO8.xInput);
END_REGION
END_FUNCTION

FUNCTION "SS1_710A1_8RTD_IO_Update" : Void   // FC11020, LAD
{ S7_Optimized_Access := 'TRUE' }
VERSION : 0.1
// stored: AutoNumber false, IsIECCheckEnabled false, SetENOAutomatically false, UDAEnableTagReadback false
BEGIN

REGION Network 1
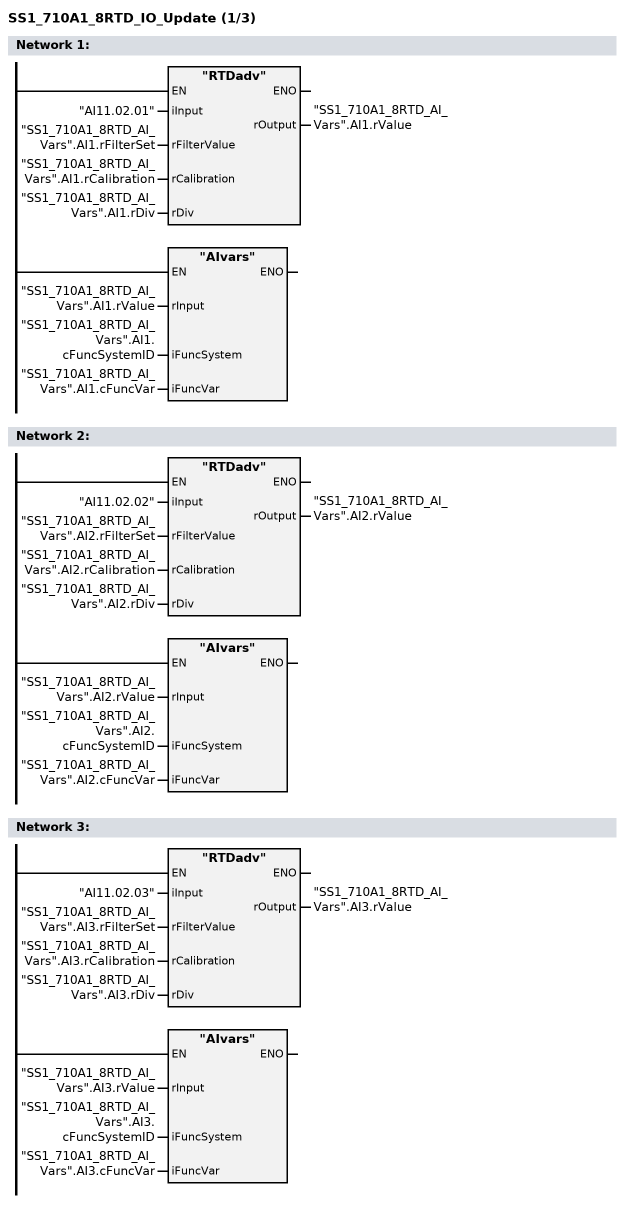
   RUNG wire#powerrail
      "RTDadv"(iInput := "AI11.02.01", rFilterValue := "SS1_710A1_8RTD_AI_Vars".AI1.rFilterSet, rCalibration := "SS1_710A1_8RTD_AI_Vars".AI1.rCalibration, rDiv := "SS1_710A1_8RTD_AI_Vars".AI1.rDiv, rOutput => "SS1_710A1_8RTD_AI_Vars".AI1.rValue)
   END_RUNG
   RUNG wire#powerrail
      "AIvars"(rInput := "SS1_710A1_8RTD_AI_Vars".AI1.rValue, iFuncSystem := "SS1_710A1_8RTD_AI_Vars".AI1.cFuncSystemID, iFuncVar := "SS1_710A1_8RTD_AI_Vars".AI1.cFuncVar)
   END_RUNG
   // the same network as SCL:
   "RTDadv"(iInput := "AI11.02.01",
            rFilterValue := "SS1_710A1_8RTD_AI_Vars".AI1.rFilterSet,
            rCalibration := "SS1_710A1_8RTD_AI_Vars".AI1.rCalibration,
            rDiv := "SS1_710A1_8RTD_AI_Vars".AI1.rDiv,
            rOutput => "SS1_710A1_8RTD_AI_Vars".AI1.rValue);
   "AIvars"(rInput := "SS1_710A1_8RTD_AI_Vars".AI1.rValue,
            iFuncSystem := "SS1_710A1_8RTD_AI_Vars".AI1.cFuncSystemID,
            iFuncVar := "SS1_710A1_8RTD_AI_Vars".AI1.cFuncVar);
END_REGION

REGION Network 2
   RUNG wire#powerrail
      "RTDadv"(iInput := "AI11.02.02", rFilterValue := "SS1_710A1_8RTD_AI_Vars".AI2.rFilterSet, rCalibration := "SS1_710A1_8RTD_AI_Vars".AI2.rCalibration, rDiv := "SS1_710A1_8RTD_AI_Vars".AI2.rDiv, rOutput => "SS1_710A1_8RTD_AI_Vars".AI2.rValue)
   END_RUNG
   RUNG wire#powerrail
      "AIvars"(rInput := "SS1_710A1_8RTD_AI_Vars".AI2.rValue, iFuncSystem := "SS1_710A1_8RTD_AI_Vars".AI2.cFuncSystemID, iFuncVar := "SS1_710A1_8RTD_AI_Vars".AI2.cFuncVar)
   END_RUNG
   // the same network as SCL:
   "RTDadv"(iInput := "AI11.02.02",
            rFilterValue := "SS1_710A1_8RTD_AI_Vars".AI2.rFilterSet,
            rCalibration := "SS1_710A1_8RTD_AI_Vars".AI2.rCalibration,
            rDiv := "SS1_710A1_8RTD_AI_Vars".AI2.rDiv,
            rOutput => "SS1_710A1_8RTD_AI_Vars".AI2.rValue);
   "AIvars"(rInput := "SS1_710A1_8RTD_AI_Vars".AI2.rValue,
            iFuncSystem := "SS1_710A1_8RTD_AI_Vars".AI2.cFuncSystemID,
            iFuncVar := "SS1_710A1_8RTD_AI_Vars".AI2.cFuncVar);
END_REGION

REGION Network 3
   RUNG wire#powerrail
      "RTDadv"(iInput := "AI11.02.03", rFilterValue := "SS1_710A1_8RTD_AI_Vars".AI3.rFilterSet, rCalibration := "SS1_710A1_8RTD_AI_Vars".AI3.rCalibration, rDiv := "SS1_710A1_8RTD_AI_Vars".AI3.rDiv, rOutput => "SS1_710A1_8RTD_AI_Vars".AI3.rValue)
   END_RUNG
   RUNG wire#powerrail
      "AIvars"(rInput := "SS1_710A1_8RTD_AI_Vars".AI3.rValue, iFuncSystem := "SS1_710A1_8RTD_AI_Vars".AI3.cFuncSystemID, iFuncVar := "SS1_710A1_8RTD_AI_Vars".AI3.cFuncVar)
   END_RUNG
   // the same network as SCL:
   "RTDadv"(iInput := "AI11.02.03",
            rFilterValue := "SS1_710A1_8RTD_AI_Vars".AI3.rFilterSet,
            rCalibration := "SS1_710A1_8RTD_AI_Vars".AI3.rCalibration,
            rDiv := "SS1_710A1_8RTD_AI_Vars".AI3.rDiv,
            rOutput => "SS1_710A1_8RTD_AI_Vars".AI3.rValue);
   "AIvars"(rInput := "SS1_710A1_8RTD_AI_Vars".AI3.rValue,
            iFuncSystem := "SS1_710A1_8RTD_AI_Vars".AI3.cFuncSystemID,
            iFuncVar := "SS1_710A1_8RTD_AI_Vars".AI3.cFuncVar);
END_REGION

REGION Network 4
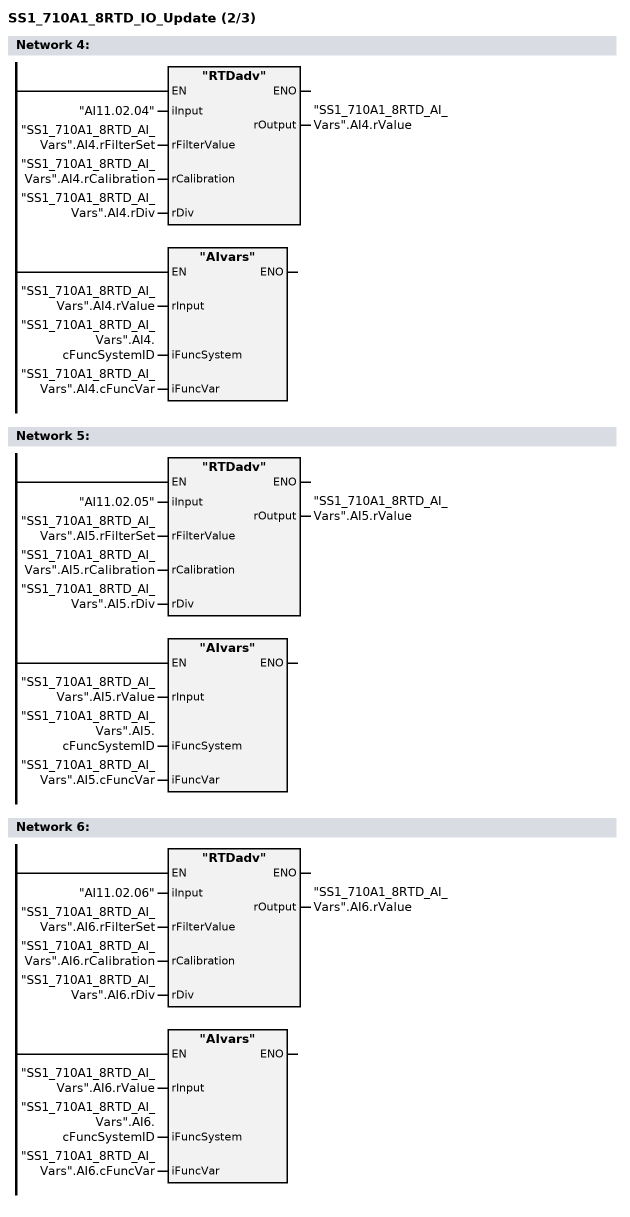
   RUNG wire#powerrail
      "RTDadv"(iInput := "AI11.02.04", rFilterValue := "SS1_710A1_8RTD_AI_Vars".AI4.rFilterSet, rCalibration := "SS1_710A1_8RTD_AI_Vars".AI4.rCalibration, rDiv := "SS1_710A1_8RTD_AI_Vars".AI4.rDiv, rOutput => "SS1_710A1_8RTD_AI_Vars".AI4.rValue)
   END_RUNG
   RUNG wire#powerrail
      "AIvars"(rInput := "SS1_710A1_8RTD_AI_Vars".AI4.rValue, iFuncSystem := "SS1_710A1_8RTD_AI_Vars".AI4.cFuncSystemID, iFuncVar := "SS1_710A1_8RTD_AI_Vars".AI4.cFuncVar)
   END_RUNG
   // the same network as SCL:
   "RTDadv"(iInput := "AI11.02.04",
            rFilterValue := "SS1_710A1_8RTD_AI_Vars".AI4.rFilterSet,
            rCalibration := "SS1_710A1_8RTD_AI_Vars".AI4.rCalibration,
            rDiv := "SS1_710A1_8RTD_AI_Vars".AI4.rDiv,
            rOutput => "SS1_710A1_8RTD_AI_Vars".AI4.rValue);
   "AIvars"(rInput := "SS1_710A1_8RTD_AI_Vars".AI4.rValue,
            iFuncSystem := "SS1_710A1_8RTD_AI_Vars".AI4.cFuncSystemID,
            iFuncVar := "SS1_710A1_8RTD_AI_Vars".AI4.cFuncVar);
END_REGION

REGION Network 5
   RUNG wire#powerrail
      "RTDadv"(iInput := "AI11.02.05", rFilterValue := "SS1_710A1_8RTD_AI_Vars".AI5.rFilterSet, rCalibration := "SS1_710A1_8RTD_AI_Vars".AI5.rCalibration, rDiv := "SS1_710A1_8RTD_AI_Vars".AI5.rDiv, rOutput => "SS1_710A1_8RTD_AI_Vars".AI5.rValue)
   END_RUNG
   RUNG wire#powerrail
      "AIvars"(rInput := "SS1_710A1_8RTD_AI_Vars".AI5.rValue, iFuncSystem := "SS1_710A1_8RTD_AI_Vars".AI5.cFuncSystemID, iFuncVar := "SS1_710A1_8RTD_AI_Vars".AI5.cFuncVar)
   END_RUNG
   // the same network as SCL:
   "RTDadv"(iInput := "AI11.02.05",
            rFilterValue := "SS1_710A1_8RTD_AI_Vars".AI5.rFilterSet,
            rCalibration := "SS1_710A1_8RTD_AI_Vars".AI5.rCalibration,
            rDiv := "SS1_710A1_8RTD_AI_Vars".AI5.rDiv,
            rOutput => "SS1_710A1_8RTD_AI_Vars".AI5.rValue);
   "AIvars"(rInput := "SS1_710A1_8RTD_AI_Vars".AI5.rValue,
            iFuncSystem := "SS1_710A1_8RTD_AI_Vars".AI5.cFuncSystemID,
            iFuncVar := "SS1_710A1_8RTD_AI_Vars".AI5.cFuncVar);
END_REGION

REGION Network 6
   RUNG wire#powerrail
      "RTDadv"(iInput := "AI11.02.06", rFilterValue := "SS1_710A1_8RTD_AI_Vars".AI6.rFilterSet, rCalibration := "SS1_710A1_8RTD_AI_Vars".AI6.rCalibration, rDiv := "SS1_710A1_8RTD_AI_Vars".AI6.rDiv, rOutput => "SS1_710A1_8RTD_AI_Vars".AI6.rValue)
   END_RUNG
   RUNG wire#powerrail
      "AIvars"(rInput := "SS1_710A1_8RTD_AI_Vars".AI6.rValue, iFuncSystem := "SS1_710A1_8RTD_AI_Vars".AI6.cFuncSystemID, iFuncVar := "SS1_710A1_8RTD_AI_Vars".AI6.cFuncVar)
   END_RUNG
   // the same network as SCL:
   "RTDadv"(iInput := "AI11.02.06",
            rFilterValue := "SS1_710A1_8RTD_AI_Vars".AI6.rFilterSet,
            rCalibration := "SS1_710A1_8RTD_AI_Vars".AI6.rCalibration,
            rDiv := "SS1_710A1_8RTD_AI_Vars".AI6.rDiv,
            rOutput => "SS1_710A1_8RTD_AI_Vars".AI6.rValue);
   "AIvars"(rInput := "SS1_710A1_8RTD_AI_Vars".AI6.rValue,
            iFuncSystem := "SS1_710A1_8RTD_AI_Vars".AI6.cFuncSystemID,
            iFuncVar := "SS1_710A1_8RTD_AI_Vars".AI6.cFuncVar);
END_REGION

REGION Network 7
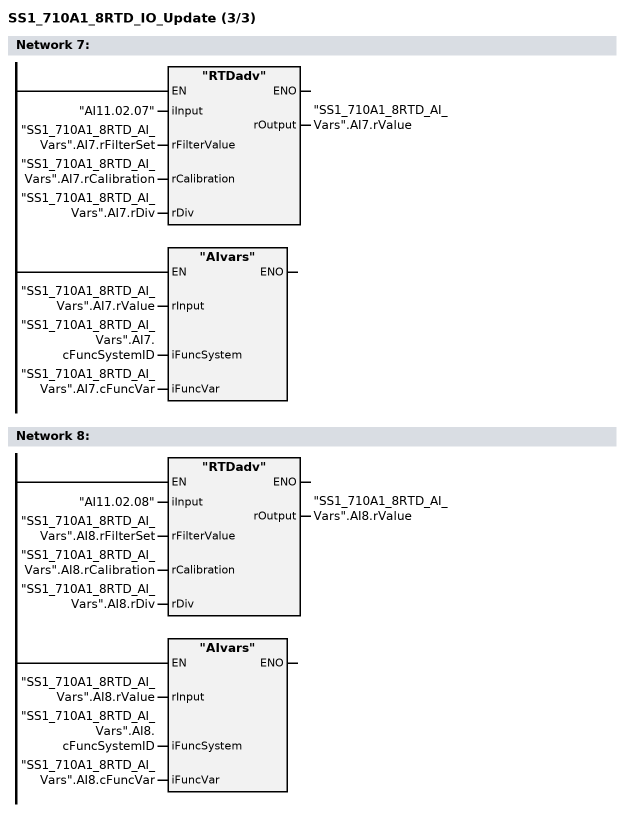
   RUNG wire#powerrail
      "RTDadv"(iInput := "AI11.02.07", rFilterValue := "SS1_710A1_8RTD_AI_Vars".AI7.rFilterSet, rCalibration := "SS1_710A1_8RTD_AI_Vars".AI7.rCalibration, rDiv := "SS1_710A1_8RTD_AI_Vars".AI7.rDiv, rOutput => "SS1_710A1_8RTD_AI_Vars".AI7.rValue)
   END_RUNG
   RUNG wire#powerrail
      "AIvars"(rInput := "SS1_710A1_8RTD_AI_Vars".AI7.rValue, iFuncSystem := "SS1_710A1_8RTD_AI_Vars".AI7.cFuncSystemID, iFuncVar := "SS1_710A1_8RTD_AI_Vars".AI7.cFuncVar)
   END_RUNG
   // the same network as SCL:
   "RTDadv"(iInput := "AI11.02.07",
            rFilterValue := "SS1_710A1_8RTD_AI_Vars".AI7.rFilterSet,
            rCalibration := "SS1_710A1_8RTD_AI_Vars".AI7.rCalibration,
            rDiv := "SS1_710A1_8RTD_AI_Vars".AI7.rDiv,
            rOutput => "SS1_710A1_8RTD_AI_Vars".AI7.rValue);
   "AIvars"(rInput := "SS1_710A1_8RTD_AI_Vars".AI7.rValue,
            iFuncSystem := "SS1_710A1_8RTD_AI_Vars".AI7.cFuncSystemID,
            iFuncVar := "SS1_710A1_8RTD_AI_Vars".AI7.cFuncVar);
END_REGION

REGION Network 8
   RUNG wire#powerrail
      "RTDadv"(iInput := "AI11.02.08", rFilterValue := "SS1_710A1_8RTD_AI_Vars".AI8.rFilterSet, rCalibration := "SS1_710A1_8RTD_AI_Vars".AI8.rCalibration, rDiv := "SS1_710A1_8RTD_AI_Vars".AI8.rDiv, rOutput => "SS1_710A1_8RTD_AI_Vars".AI8.rValue)
   END_RUNG
   RUNG wire#powerrail
      "AIvars"(rInput := "SS1_710A1_8RTD_AI_Vars".AI8.rValue, iFuncSystem := "SS1_710A1_8RTD_AI_Vars".AI8.cFuncSystemID, iFuncVar := "SS1_710A1_8RTD_AI_Vars".AI8.cFuncVar)
   END_RUNG
   // the same network as SCL:
   "RTDadv"(iInput := "AI11.02.08",
            rFilterValue := "SS1_710A1_8RTD_AI_Vars".AI8.rFilterSet,
            rCalibration := "SS1_710A1_8RTD_AI_Vars".AI8.rCalibration,
            rDiv := "SS1_710A1_8RTD_AI_Vars".AI8.rDiv,
            rOutput => "SS1_710A1_8RTD_AI_Vars".AI8.rValue);
   "AIvars"(rInput := "SS1_710A1_8RTD_AI_Vars".AI8.rValue,
            iFuncSystem := "SS1_710A1_8RTD_AI_Vars".AI8.cFuncSystemID,
            iFuncVar := "SS1_710A1_8RTD_AI_Vars".AI8.cFuncVar);
END_REGION
END_FUNCTION

FUNCTION "SS1_730A1_4AO_IO_Update" : Void   // FC11040, LAD
{ S7_Optimized_Access := 'TRUE' }
VERSION : 0.1
// stored: AutoNumber false, IsIECCheckEnabled false, SetENOAutomatically false, UDAEnableTagReadback false
BEGIN

REGION Network 1: AO0
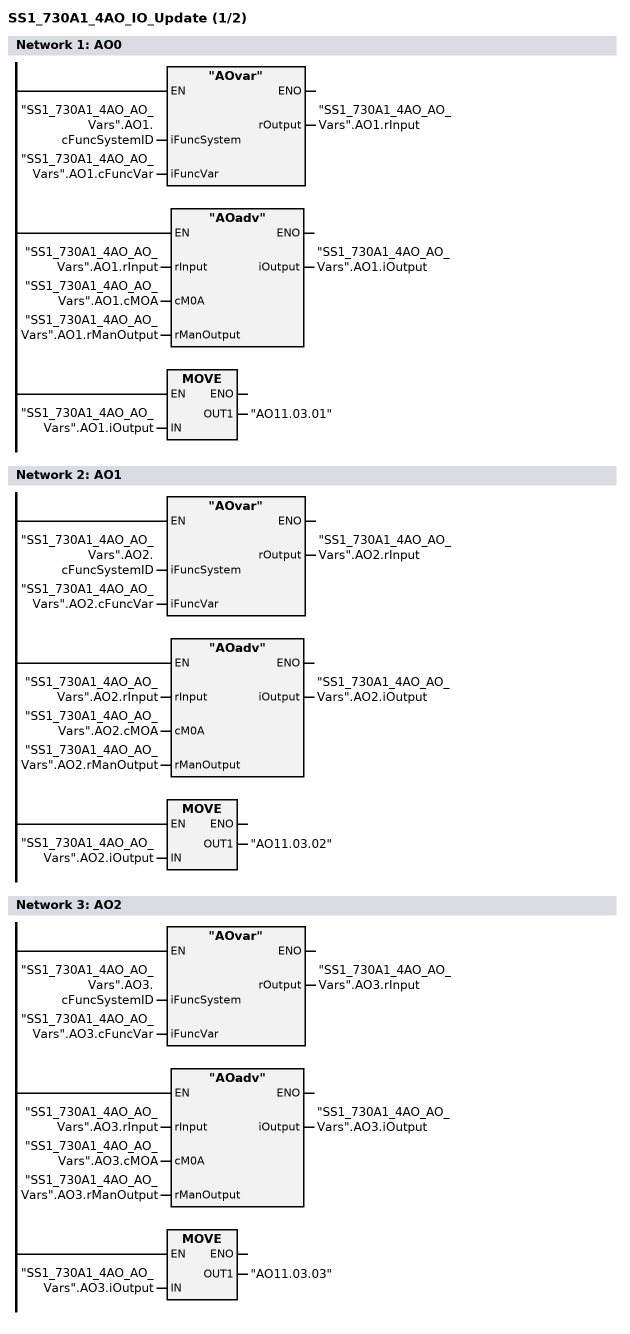
   RUNG wire#powerrail
      "AOvar"(iFuncSystem := "SS1_730A1_4AO_AO_Vars".AO1.cFuncSystemID, iFuncVar := "SS1_730A1_4AO_AO_Vars".AO1.cFuncVar, rOutput => "SS1_730A1_4AO_AO_Vars".AO1.rInput)
   END_RUNG
   RUNG wire#powerrail
      "AOadv"(rInput := "SS1_730A1_4AO_AO_Vars".AO1.rInput, cM0A := "SS1_730A1_4AO_AO_Vars".AO1.cMOA, rManOutput := "SS1_730A1_4AO_AO_Vars".AO1.rManOutput, iOutput => "SS1_730A1_4AO_AO_Vars".AO1.iOutput)
   END_RUNG
   RUNG wire#powerrail
      Move(in := "SS1_730A1_4AO_AO_Vars".AO1.iOutput, out1 => "AO11.03.01")
   END_RUNG
   // the same network as SCL:
   "AOvar"(iFuncSystem := "SS1_730A1_4AO_AO_Vars".AO1.cFuncSystemID,
           iFuncVar := "SS1_730A1_4AO_AO_Vars".AO1.cFuncVar,
           rOutput => "SS1_730A1_4AO_AO_Vars".AO1.rInput);
   "AOadv"(rInput := "SS1_730A1_4AO_AO_Vars".AO1.rInput,
           cM0A := "SS1_730A1_4AO_AO_Vars".AO1.cMOA,
           rManOutput := "SS1_730A1_4AO_AO_Vars".AO1.rManOutput,
           iOutput => "SS1_730A1_4AO_AO_Vars".AO1.iOutput);
   "AO11.03.01" := "SS1_730A1_4AO_AO_Vars".AO1.iOutput;
END_REGION

REGION Network 2: AO1
   RUNG wire#powerrail
      "AOvar"(iFuncSystem := "SS1_730A1_4AO_AO_Vars".AO2.cFuncSystemID, iFuncVar := "SS1_730A1_4AO_AO_Vars".AO2.cFuncVar, rOutput => "SS1_730A1_4AO_AO_Vars".AO2.rInput)
   END_RUNG
   RUNG wire#powerrail
      "AOadv"(rInput := "SS1_730A1_4AO_AO_Vars".AO2.rInput, cM0A := "SS1_730A1_4AO_AO_Vars".AO2.cMOA, rManOutput := "SS1_730A1_4AO_AO_Vars".AO2.rManOutput, iOutput => "SS1_730A1_4AO_AO_Vars".AO2.iOutput)
   END_RUNG
   RUNG wire#powerrail
      Move(in := "SS1_730A1_4AO_AO_Vars".AO2.iOutput, out1 => "AO11.03.02")
   END_RUNG
   // the same network as SCL:
   "AOvar"(iFuncSystem := "SS1_730A1_4AO_AO_Vars".AO2.cFuncSystemID,
           iFuncVar := "SS1_730A1_4AO_AO_Vars".AO2.cFuncVar,
           rOutput => "SS1_730A1_4AO_AO_Vars".AO2.rInput);
   "AOadv"(rInput := "SS1_730A1_4AO_AO_Vars".AO2.rInput,
           cM0A := "SS1_730A1_4AO_AO_Vars".AO2.cMOA,
           rManOutput := "SS1_730A1_4AO_AO_Vars".AO2.rManOutput,
           iOutput => "SS1_730A1_4AO_AO_Vars".AO2.iOutput);
   "AO11.03.02" := "SS1_730A1_4AO_AO_Vars".AO2.iOutput;
END_REGION

REGION Network 3: AO2
   RUNG wire#powerrail
      "AOvar"(iFuncSystem := "SS1_730A1_4AO_AO_Vars".AO3.cFuncSystemID, iFuncVar := "SS1_730A1_4AO_AO_Vars".AO3.cFuncVar, rOutput => "SS1_730A1_4AO_AO_Vars".AO3.rInput)
   END_RUNG
   RUNG wire#powerrail
      "AOadv"(rInput := "SS1_730A1_4AO_AO_Vars".AO3.rInput, cM0A := "SS1_730A1_4AO_AO_Vars".AO3.cMOA, rManOutput := "SS1_730A1_4AO_AO_Vars".AO3.rManOutput, iOutput => "SS1_730A1_4AO_AO_Vars".AO3.iOutput)
   END_RUNG
   RUNG wire#powerrail
      Move(in := "SS1_730A1_4AO_AO_Vars".AO3.iOutput, out1 => "AO11.03.03")
   END_RUNG
   // the same network as SCL:
   "AOvar"(iFuncSystem := "SS1_730A1_4AO_AO_Vars".AO3.cFuncSystemID,
           iFuncVar := "SS1_730A1_4AO_AO_Vars".AO3.cFuncVar,
           rOutput => "SS1_730A1_4AO_AO_Vars".AO3.rInput);
   "AOadv"(rInput := "SS1_730A1_4AO_AO_Vars".AO3.rInput,
           cM0A := "SS1_730A1_4AO_AO_Vars".AO3.cMOA,
           rManOutput := "SS1_730A1_4AO_AO_Vars".AO3.rManOutput,
           iOutput => "SS1_730A1_4AO_AO_Vars".AO3.iOutput);
   "AO11.03.03" := "SS1_730A1_4AO_AO_Vars".AO3.iOutput;
END_REGION

REGION Network 4: AO3
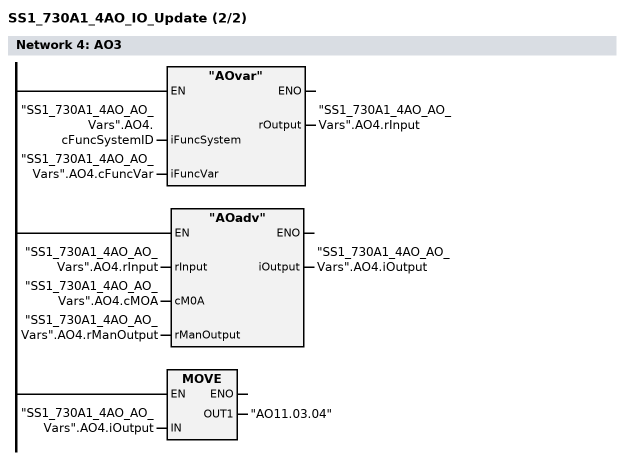
   RUNG wire#powerrail
      "AOvar"(iFuncSystem := "SS1_730A1_4AO_AO_Vars".AO4.cFuncSystemID, iFuncVar := "SS1_730A1_4AO_AO_Vars".AO4.cFuncVar, rOutput => "SS1_730A1_4AO_AO_Vars".AO4.rInput)
   END_RUNG
   RUNG wire#powerrail
      "AOadv"(rInput := "SS1_730A1_4AO_AO_Vars".AO4.rInput, cM0A := "SS1_730A1_4AO_AO_Vars".AO4.cMOA, rManOutput := "SS1_730A1_4AO_AO_Vars".AO4.rManOutput, iOutput => "SS1_730A1_4AO_AO_Vars".AO4.iOutput)
   END_RUNG
   RUNG wire#powerrail
      Move(in := "SS1_730A1_4AO_AO_Vars".AO4.iOutput, out1 => "AO11.03.04")
   END_RUNG
   // the same network as SCL:
   "AOvar"(iFuncSystem := "SS1_730A1_4AO_AO_Vars".AO4.cFuncSystemID,
           iFuncVar := "SS1_730A1_4AO_AO_Vars".AO4.cFuncVar,
           rOutput => "SS1_730A1_4AO_AO_Vars".AO4.rInput);
   "AOadv"(rInput := "SS1_730A1_4AO_AO_Vars".AO4.rInput,
           cM0A := "SS1_730A1_4AO_AO_Vars".AO4.cMOA,
           rManOutput := "SS1_730A1_4AO_AO_Vars".AO4.rManOutput,
           iOutput => "SS1_730A1_4AO_AO_Vars".AO4.iOutput);
   "AO11.03.04" := "SS1_730A1_4AO_AO_Vars".AO4.iOutput;
END_REGION
END_FUNCTION

FUNCTION "SS1_750A1_16DI_IO_Update" : Void   // FC11050, LAD
{ S7_Optimized_Access := 'TRUE' }
VERSION : 0.1
// stored: AutoNumber false, IsIECCheckEnabled false, SetENOAutomatically false, UDAEnableTagReadback false
BEGIN

REGION Network 1: DIa0
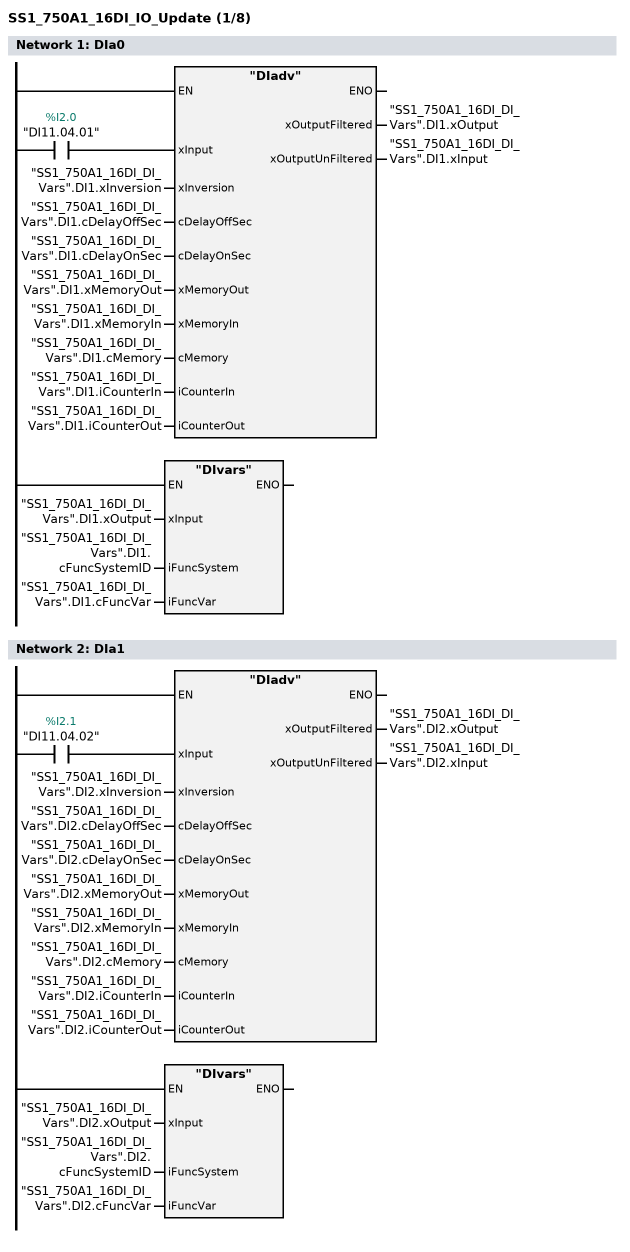
   RUNG wire#powerrail
      "DIadv"(xInput := wire#w1, xInversion := "SS1_750A1_16DI_DI_Vars".DI1.xInversion, cDelayOffSec := "SS1_750A1_16DI_DI_Vars".DI1.cDelayOffSec, cDelayOnSec := "SS1_750A1_16DI_DI_Vars".DI1.cDelayOnSec, xMemoryOut := "SS1_750A1_16DI_DI_Vars".DI1.xMemoryOut, xMemoryIn := "SS1_750A1_16DI_DI_Vars".DI1.xMemoryIn, cMemory := "SS1_750A1_16DI_DI_Vars".DI1.cMemory, iCounterIn := "SS1_750A1_16DI_DI_Vars".DI1.iCounterIn, iCounterOut := "SS1_750A1_16DI_DI_Vars".DI1.iCounterOut, xOutputFiltered => "SS1_750A1_16DI_DI_Vars".DI1.xOutput, xOutputUnFiltered => "SS1_750A1_16DI_DI_Vars".DI1.xInput)
   END_RUNG
   RUNG wire#powerrail
      Contact( "DI11.04.01" )
   END_RUNG wire#w1
   RUNG wire#powerrail
      "DIvars"(xInput := "SS1_750A1_16DI_DI_Vars".DI1.xOutput, iFuncSystem := "SS1_750A1_16DI_DI_Vars".DI1.cFuncSystemID, iFuncVar := "SS1_750A1_16DI_DI_Vars".DI1.cFuncVar)
   END_RUNG
   // the same network as SCL:
   "DIadv"(xInput := "DI11.04.01",
           xInversion := "SS1_750A1_16DI_DI_Vars".DI1.xInversion,
           cDelayOffSec := "SS1_750A1_16DI_DI_Vars".DI1.cDelayOffSec,
           cDelayOnSec := "SS1_750A1_16DI_DI_Vars".DI1.cDelayOnSec,
           xMemoryOut := "SS1_750A1_16DI_DI_Vars".DI1.xMemoryOut,
           xMemoryIn := "SS1_750A1_16DI_DI_Vars".DI1.xMemoryIn,
           cMemory := "SS1_750A1_16DI_DI_Vars".DI1.cMemory,
           iCounterIn := "SS1_750A1_16DI_DI_Vars".DI1.iCounterIn,
           iCounterOut := "SS1_750A1_16DI_DI_Vars".DI1.iCounterOut,
           xOutputFiltered => "SS1_750A1_16DI_DI_Vars".DI1.xOutput,
           xOutputUnFiltered => "SS1_750A1_16DI_DI_Vars".DI1.xInput);
   "DIvars"(xInput := "SS1_750A1_16DI_DI_Vars".DI1.xOutput,
            iFuncSystem := "SS1_750A1_16DI_DI_Vars".DI1.cFuncSystemID,
            iFuncVar := "SS1_750A1_16DI_DI_Vars".DI1.cFuncVar);
END_REGION

REGION Network 2: DIa1
   RUNG wire#powerrail
      "DIadv"(xInput := wire#w1, xInversion := "SS1_750A1_16DI_DI_Vars".DI2.xInversion, cDelayOffSec := "SS1_750A1_16DI_DI_Vars".DI2.cDelayOffSec, cDelayOnSec := "SS1_750A1_16DI_DI_Vars".DI2.cDelayOnSec, xMemoryOut := "SS1_750A1_16DI_DI_Vars".DI2.xMemoryOut, xMemoryIn := "SS1_750A1_16DI_DI_Vars".DI2.xMemoryIn, cMemory := "SS1_750A1_16DI_DI_Vars".DI2.cMemory, iCounterIn := "SS1_750A1_16DI_DI_Vars".DI2.iCounterIn, iCounterOut := "SS1_750A1_16DI_DI_Vars".DI2.iCounterOut, xOutputFiltered => "SS1_750A1_16DI_DI_Vars".DI2.xOutput, xOutputUnFiltered => "SS1_750A1_16DI_DI_Vars".DI2.xInput)
   END_RUNG
   RUNG wire#powerrail
      Contact( "DI11.04.02" )
   END_RUNG wire#w1
   RUNG wire#powerrail
      "DIvars"(xInput := "SS1_750A1_16DI_DI_Vars".DI2.xOutput, iFuncSystem := "SS1_750A1_16DI_DI_Vars".DI2.cFuncSystemID, iFuncVar := "SS1_750A1_16DI_DI_Vars".DI2.cFuncVar)
   END_RUNG
   // the same network as SCL:
   "DIadv"(xInput := "DI11.04.02",
           xInversion := "SS1_750A1_16DI_DI_Vars".DI2.xInversion,
           cDelayOffSec := "SS1_750A1_16DI_DI_Vars".DI2.cDelayOffSec,
           cDelayOnSec := "SS1_750A1_16DI_DI_Vars".DI2.cDelayOnSec,
           xMemoryOut := "SS1_750A1_16DI_DI_Vars".DI2.xMemoryOut,
           xMemoryIn := "SS1_750A1_16DI_DI_Vars".DI2.xMemoryIn,
           cMemory := "SS1_750A1_16DI_DI_Vars".DI2.cMemory,
           iCounterIn := "SS1_750A1_16DI_DI_Vars".DI2.iCounterIn,
           iCounterOut := "SS1_750A1_16DI_DI_Vars".DI2.iCounterOut,
           xOutputFiltered => "SS1_750A1_16DI_DI_Vars".DI2.xOutput,
           xOutputUnFiltered => "SS1_750A1_16DI_DI_Vars".DI2.xInput);
   "DIvars"(xInput := "SS1_750A1_16DI_DI_Vars".DI2.xOutput,
            iFuncSystem := "SS1_750A1_16DI_DI_Vars".DI2.cFuncSystemID,
            iFuncVar := "SS1_750A1_16DI_DI_Vars".DI2.cFuncVar);
END_REGION

REGION Network 3: DIa2
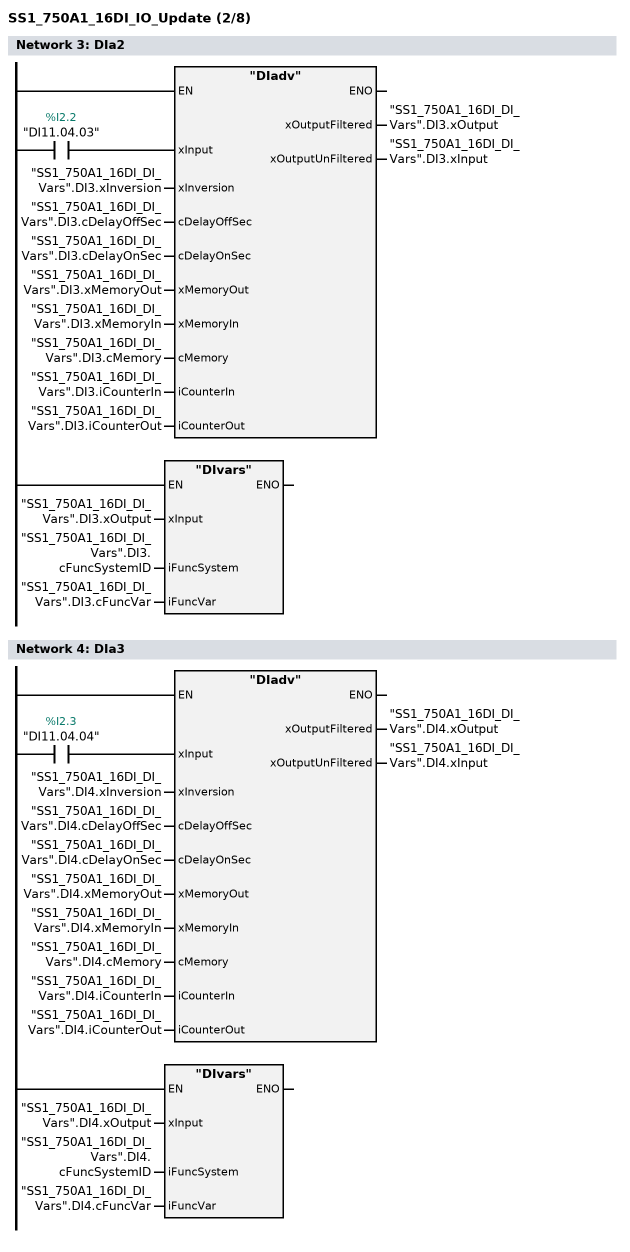
   RUNG wire#powerrail
      "DIadv"(xInput := wire#w1, xInversion := "SS1_750A1_16DI_DI_Vars".DI3.xInversion, cDelayOffSec := "SS1_750A1_16DI_DI_Vars".DI3.cDelayOffSec, cDelayOnSec := "SS1_750A1_16DI_DI_Vars".DI3.cDelayOnSec, xMemoryOut := "SS1_750A1_16DI_DI_Vars".DI3.xMemoryOut, xMemoryIn := "SS1_750A1_16DI_DI_Vars".DI3.xMemoryIn, cMemory := "SS1_750A1_16DI_DI_Vars".DI3.cMemory, iCounterIn := "SS1_750A1_16DI_DI_Vars".DI3.iCounterIn, iCounterOut := "SS1_750A1_16DI_DI_Vars".DI3.iCounterOut, xOutputFiltered => "SS1_750A1_16DI_DI_Vars".DI3.xOutput, xOutputUnFiltered => "SS1_750A1_16DI_DI_Vars".DI3.xInput)
   END_RUNG
   RUNG wire#powerrail
      Contact( "DI11.04.03" )
   END_RUNG wire#w1
   RUNG wire#powerrail
      "DIvars"(xInput := "SS1_750A1_16DI_DI_Vars".DI3.xOutput, iFuncSystem := "SS1_750A1_16DI_DI_Vars".DI3.cFuncSystemID, iFuncVar := "SS1_750A1_16DI_DI_Vars".DI3.cFuncVar)
   END_RUNG
   // the same network as SCL:
   "DIadv"(xInput := "DI11.04.03",
           xInversion := "SS1_750A1_16DI_DI_Vars".DI3.xInversion,
           cDelayOffSec := "SS1_750A1_16DI_DI_Vars".DI3.cDelayOffSec,
           cDelayOnSec := "SS1_750A1_16DI_DI_Vars".DI3.cDelayOnSec,
           xMemoryOut := "SS1_750A1_16DI_DI_Vars".DI3.xMemoryOut,
           xMemoryIn := "SS1_750A1_16DI_DI_Vars".DI3.xMemoryIn,
           cMemory := "SS1_750A1_16DI_DI_Vars".DI3.cMemory,
           iCounterIn := "SS1_750A1_16DI_DI_Vars".DI3.iCounterIn,
           iCounterOut := "SS1_750A1_16DI_DI_Vars".DI3.iCounterOut,
           xOutputFiltered => "SS1_750A1_16DI_DI_Vars".DI3.xOutput,
           xOutputUnFiltered => "SS1_750A1_16DI_DI_Vars".DI3.xInput);
   "DIvars"(xInput := "SS1_750A1_16DI_DI_Vars".DI3.xOutput,
            iFuncSystem := "SS1_750A1_16DI_DI_Vars".DI3.cFuncSystemID,
            iFuncVar := "SS1_750A1_16DI_DI_Vars".DI3.cFuncVar);
END_REGION

REGION Network 4: DIa3
   RUNG wire#powerrail
      "DIadv"(xInput := wire#w1, xInversion := "SS1_750A1_16DI_DI_Vars".DI4.xInversion, cDelayOffSec := "SS1_750A1_16DI_DI_Vars".DI4.cDelayOffSec, cDelayOnSec := "SS1_750A1_16DI_DI_Vars".DI4.cDelayOnSec, xMemoryOut := "SS1_750A1_16DI_DI_Vars".DI4.xMemoryOut, xMemoryIn := "SS1_750A1_16DI_DI_Vars".DI4.xMemoryIn, cMemory := "SS1_750A1_16DI_DI_Vars".DI4.cMemory, iCounterIn := "SS1_750A1_16DI_DI_Vars".DI4.iCounterIn, iCounterOut := "SS1_750A1_16DI_DI_Vars".DI4.iCounterOut, xOutputFiltered => "SS1_750A1_16DI_DI_Vars".DI4.xOutput, xOutputUnFiltered => "SS1_750A1_16DI_DI_Vars".DI4.xInput)
   END_RUNG
   RUNG wire#powerrail
      Contact( "DI11.04.04" )
   END_RUNG wire#w1
   RUNG wire#powerrail
      "DIvars"(xInput := "SS1_750A1_16DI_DI_Vars".DI4.xOutput, iFuncSystem := "SS1_750A1_16DI_DI_Vars".DI4.cFuncSystemID, iFuncVar := "SS1_750A1_16DI_DI_Vars".DI4.cFuncVar)
   END_RUNG
   // the same network as SCL:
   "DIadv"(xInput := "DI11.04.04",
           xInversion := "SS1_750A1_16DI_DI_Vars".DI4.xInversion,
           cDelayOffSec := "SS1_750A1_16DI_DI_Vars".DI4.cDelayOffSec,
           cDelayOnSec := "SS1_750A1_16DI_DI_Vars".DI4.cDelayOnSec,
           xMemoryOut := "SS1_750A1_16DI_DI_Vars".DI4.xMemoryOut,
           xMemoryIn := "SS1_750A1_16DI_DI_Vars".DI4.xMemoryIn,
           cMemory := "SS1_750A1_16DI_DI_Vars".DI4.cMemory,
           iCounterIn := "SS1_750A1_16DI_DI_Vars".DI4.iCounterIn,
           iCounterOut := "SS1_750A1_16DI_DI_Vars".DI4.iCounterOut,
           xOutputFiltered => "SS1_750A1_16DI_DI_Vars".DI4.xOutput,
           xOutputUnFiltered => "SS1_750A1_16DI_DI_Vars".DI4.xInput);
   "DIvars"(xInput := "SS1_750A1_16DI_DI_Vars".DI4.xOutput,
            iFuncSystem := "SS1_750A1_16DI_DI_Vars".DI4.cFuncSystemID,
            iFuncVar := "SS1_750A1_16DI_DI_Vars".DI4.cFuncVar);
END_REGION

REGION Network 5: DIa4
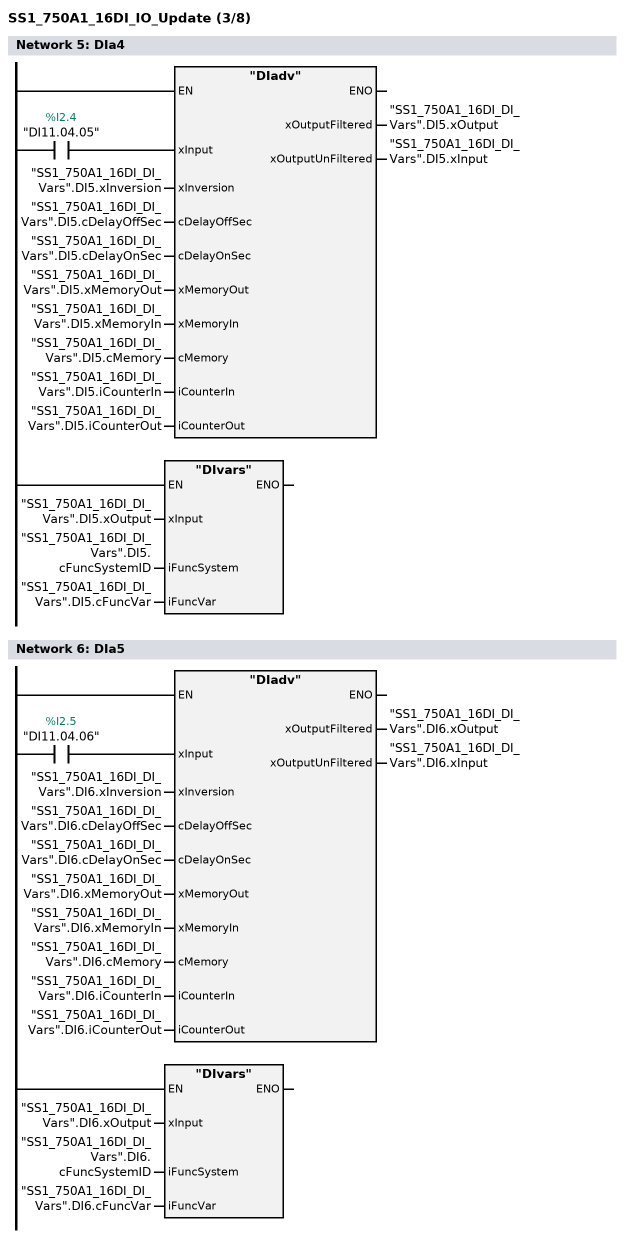
   RUNG wire#powerrail
      "DIadv"(xInput := wire#w1, xInversion := "SS1_750A1_16DI_DI_Vars".DI5.xInversion, cDelayOffSec := "SS1_750A1_16DI_DI_Vars".DI5.cDelayOffSec, cDelayOnSec := "SS1_750A1_16DI_DI_Vars".DI5.cDelayOnSec, xMemoryOut := "SS1_750A1_16DI_DI_Vars".DI5.xMemoryOut, xMemoryIn := "SS1_750A1_16DI_DI_Vars".DI5.xMemoryIn, cMemory := "SS1_750A1_16DI_DI_Vars".DI5.cMemory, iCounterIn := "SS1_750A1_16DI_DI_Vars".DI5.iCounterIn, iCounterOut := "SS1_750A1_16DI_DI_Vars".DI5.iCounterOut, xOutputFiltered => "SS1_750A1_16DI_DI_Vars".DI5.xOutput, xOutputUnFiltered => "SS1_750A1_16DI_DI_Vars".DI5.xInput)
   END_RUNG
   RUNG wire#powerrail
      Contact( "DI11.04.05" )
   END_RUNG wire#w1
   RUNG wire#powerrail
      "DIvars"(xInput := "SS1_750A1_16DI_DI_Vars".DI5.xOutput, iFuncSystem := "SS1_750A1_16DI_DI_Vars".DI5.cFuncSystemID, iFuncVar := "SS1_750A1_16DI_DI_Vars".DI5.cFuncVar)
   END_RUNG
   // the same network as SCL:
   "DIadv"(xInput := "DI11.04.05",
           xInversion := "SS1_750A1_16DI_DI_Vars".DI5.xInversion,
           cDelayOffSec := "SS1_750A1_16DI_DI_Vars".DI5.cDelayOffSec,
           cDelayOnSec := "SS1_750A1_16DI_DI_Vars".DI5.cDelayOnSec,
           xMemoryOut := "SS1_750A1_16DI_DI_Vars".DI5.xMemoryOut,
           xMemoryIn := "SS1_750A1_16DI_DI_Vars".DI5.xMemoryIn,
           cMemory := "SS1_750A1_16DI_DI_Vars".DI5.cMemory,
           iCounterIn := "SS1_750A1_16DI_DI_Vars".DI5.iCounterIn,
           iCounterOut := "SS1_750A1_16DI_DI_Vars".DI5.iCounterOut,
           xOutputFiltered => "SS1_750A1_16DI_DI_Vars".DI5.xOutput,
           xOutputUnFiltered => "SS1_750A1_16DI_DI_Vars".DI5.xInput);
   "DIvars"(xInput := "SS1_750A1_16DI_DI_Vars".DI5.xOutput,
            iFuncSystem := "SS1_750A1_16DI_DI_Vars".DI5.cFuncSystemID,
            iFuncVar := "SS1_750A1_16DI_DI_Vars".DI5.cFuncVar);
END_REGION

REGION Network 6: DIa5
   RUNG wire#powerrail
      "DIadv"(xInput := wire#w1, xInversion := "SS1_750A1_16DI_DI_Vars".DI6.xInversion, cDelayOffSec := "SS1_750A1_16DI_DI_Vars".DI6.cDelayOffSec, cDelayOnSec := "SS1_750A1_16DI_DI_Vars".DI6.cDelayOnSec, xMemoryOut := "SS1_750A1_16DI_DI_Vars".DI6.xMemoryOut, xMemoryIn := "SS1_750A1_16DI_DI_Vars".DI6.xMemoryIn, cMemory := "SS1_750A1_16DI_DI_Vars".DI6.cMemory, iCounterIn := "SS1_750A1_16DI_DI_Vars".DI6.iCounterIn, iCounterOut := "SS1_750A1_16DI_DI_Vars".DI6.iCounterOut, xOutputFiltered => "SS1_750A1_16DI_DI_Vars".DI6.xOutput, xOutputUnFiltered => "SS1_750A1_16DI_DI_Vars".DI6.xInput)
   END_RUNG
   RUNG wire#powerrail
      Contact( "DI11.04.06" )
   END_RUNG wire#w1
   RUNG wire#powerrail
      "DIvars"(xInput := "SS1_750A1_16DI_DI_Vars".DI6.xOutput, iFuncSystem := "SS1_750A1_16DI_DI_Vars".DI6.cFuncSystemID, iFuncVar := "SS1_750A1_16DI_DI_Vars".DI6.cFuncVar)
   END_RUNG
   // the same network as SCL:
   "DIadv"(xInput := "DI11.04.06",
           xInversion := "SS1_750A1_16DI_DI_Vars".DI6.xInversion,
           cDelayOffSec := "SS1_750A1_16DI_DI_Vars".DI6.cDelayOffSec,
           cDelayOnSec := "SS1_750A1_16DI_DI_Vars".DI6.cDelayOnSec,
           xMemoryOut := "SS1_750A1_16DI_DI_Vars".DI6.xMemoryOut,
           xMemoryIn := "SS1_750A1_16DI_DI_Vars".DI6.xMemoryIn,
           cMemory := "SS1_750A1_16DI_DI_Vars".DI6.cMemory,
           iCounterIn := "SS1_750A1_16DI_DI_Vars".DI6.iCounterIn,
           iCounterOut := "SS1_750A1_16DI_DI_Vars".DI6.iCounterOut,
           xOutputFiltered => "SS1_750A1_16DI_DI_Vars".DI6.xOutput,
           xOutputUnFiltered => "SS1_750A1_16DI_DI_Vars".DI6.xInput);
   "DIvars"(xInput := "SS1_750A1_16DI_DI_Vars".DI6.xOutput,
            iFuncSystem := "SS1_750A1_16DI_DI_Vars".DI6.cFuncSystemID,
            iFuncVar := "SS1_750A1_16DI_DI_Vars".DI6.cFuncVar);
END_REGION

REGION Network 7: DIa6
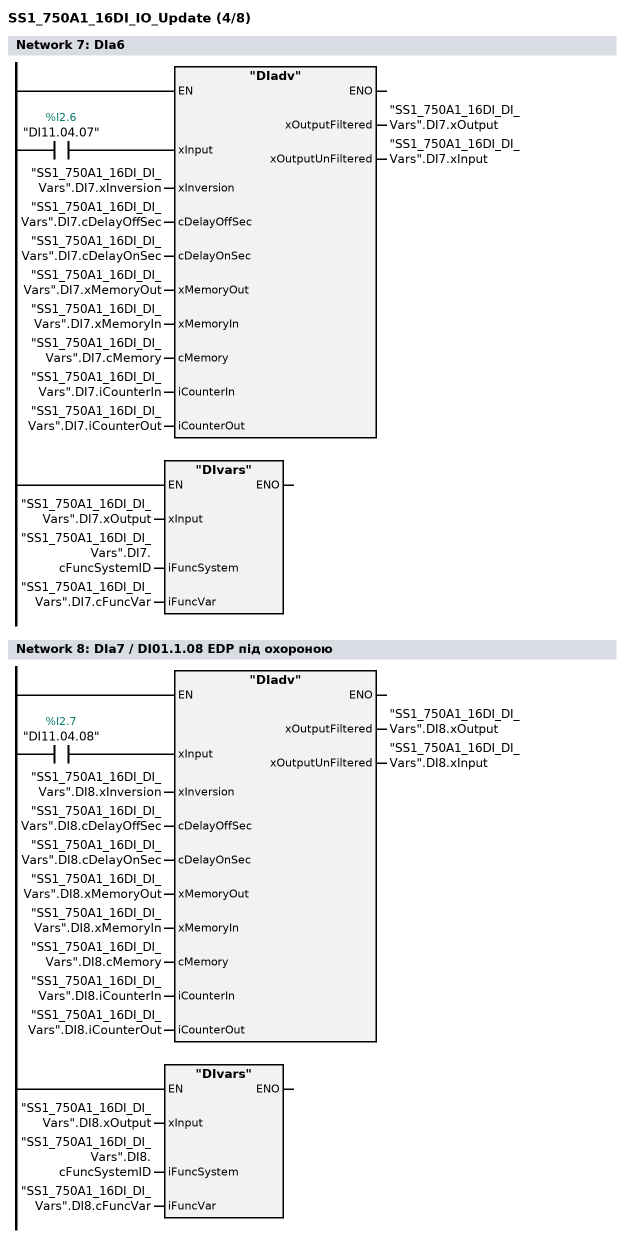
   RUNG wire#powerrail
      "DIadv"(xInput := wire#w1, xInversion := "SS1_750A1_16DI_DI_Vars".DI7.xInversion, cDelayOffSec := "SS1_750A1_16DI_DI_Vars".DI7.cDelayOffSec, cDelayOnSec := "SS1_750A1_16DI_DI_Vars".DI7.cDelayOnSec, xMemoryOut := "SS1_750A1_16DI_DI_Vars".DI7.xMemoryOut, xMemoryIn := "SS1_750A1_16DI_DI_Vars".DI7.xMemoryIn, cMemory := "SS1_750A1_16DI_DI_Vars".DI7.cMemory, iCounterIn := "SS1_750A1_16DI_DI_Vars".DI7.iCounterIn, iCounterOut := "SS1_750A1_16DI_DI_Vars".DI7.iCounterOut, xOutputFiltered => "SS1_750A1_16DI_DI_Vars".DI7.xOutput, xOutputUnFiltered => "SS1_750A1_16DI_DI_Vars".DI7.xInput)
   END_RUNG
   RUNG wire#powerrail
      Contact( "DI11.04.07" )
   END_RUNG wire#w1
   RUNG wire#powerrail
      "DIvars"(xInput := "SS1_750A1_16DI_DI_Vars".DI7.xOutput, iFuncSystem := "SS1_750A1_16DI_DI_Vars".DI7.cFuncSystemID, iFuncVar := "SS1_750A1_16DI_DI_Vars".DI7.cFuncVar)
   END_RUNG
   // the same network as SCL:
   "DIadv"(xInput := "DI11.04.07",
           xInversion := "SS1_750A1_16DI_DI_Vars".DI7.xInversion,
           cDelayOffSec := "SS1_750A1_16DI_DI_Vars".DI7.cDelayOffSec,
           cDelayOnSec := "SS1_750A1_16DI_DI_Vars".DI7.cDelayOnSec,
           xMemoryOut := "SS1_750A1_16DI_DI_Vars".DI7.xMemoryOut,
           xMemoryIn := "SS1_750A1_16DI_DI_Vars".DI7.xMemoryIn,
           cMemory := "SS1_750A1_16DI_DI_Vars".DI7.cMemory,
           iCounterIn := "SS1_750A1_16DI_DI_Vars".DI7.iCounterIn,
           iCounterOut := "SS1_750A1_16DI_DI_Vars".DI7.iCounterOut,
           xOutputFiltered => "SS1_750A1_16DI_DI_Vars".DI7.xOutput,
           xOutputUnFiltered => "SS1_750A1_16DI_DI_Vars".DI7.xInput);
   "DIvars"(xInput := "SS1_750A1_16DI_DI_Vars".DI7.xOutput,
            iFuncSystem := "SS1_750A1_16DI_DI_Vars".DI7.cFuncSystemID,
            iFuncVar := "SS1_750A1_16DI_DI_Vars".DI7.cFuncVar);
END_REGION

REGION Network 8: DIa7 / DI01.1.08 EDP під охороною
   RUNG wire#powerrail
      "DIadv"(xInput := wire#w1, xInversion := "SS1_750A1_16DI_DI_Vars".DI8.xInversion, cDelayOffSec := "SS1_750A1_16DI_DI_Vars".DI8.cDelayOffSec, cDelayOnSec := "SS1_750A1_16DI_DI_Vars".DI8.cDelayOnSec, xMemoryOut := "SS1_750A1_16DI_DI_Vars".DI8.xMemoryOut, xMemoryIn := "SS1_750A1_16DI_DI_Vars".DI8.xMemoryIn, cMemory := "SS1_750A1_16DI_DI_Vars".DI8.cMemory, iCounterIn := "SS1_750A1_16DI_DI_Vars".DI8.iCounterIn, iCounterOut := "SS1_750A1_16DI_DI_Vars".DI8.iCounterOut, xOutputFiltered => "SS1_750A1_16DI_DI_Vars".DI8.xOutput, xOutputUnFiltered => "SS1_750A1_16DI_DI_Vars".DI8.xInput)
   END_RUNG
   RUNG wire#powerrail
      Contact( "DI11.04.08" )
   END_RUNG wire#w1
   RUNG wire#powerrail
      "DIvars"(xInput := "SS1_750A1_16DI_DI_Vars".DI8.xOutput, iFuncSystem := "SS1_750A1_16DI_DI_Vars".DI8.cFuncSystemID, iFuncVar := "SS1_750A1_16DI_DI_Vars".DI8.cFuncVar)
   END_RUNG
   // the same network as SCL:
   "DIadv"(xInput := "DI11.04.08",
           xInversion := "SS1_750A1_16DI_DI_Vars".DI8.xInversion,
           cDelayOffSec := "SS1_750A1_16DI_DI_Vars".DI8.cDelayOffSec,
           cDelayOnSec := "SS1_750A1_16DI_DI_Vars".DI8.cDelayOnSec,
           xMemoryOut := "SS1_750A1_16DI_DI_Vars".DI8.xMemoryOut,
           xMemoryIn := "SS1_750A1_16DI_DI_Vars".DI8.xMemoryIn,
           cMemory := "SS1_750A1_16DI_DI_Vars".DI8.cMemory,
           iCounterIn := "SS1_750A1_16DI_DI_Vars".DI8.iCounterIn,
           iCounterOut := "SS1_750A1_16DI_DI_Vars".DI8.iCounterOut,
           xOutputFiltered => "SS1_750A1_16DI_DI_Vars".DI8.xOutput,
           xOutputUnFiltered => "SS1_750A1_16DI_DI_Vars".DI8.xInput);
   "DIvars"(xInput := "SS1_750A1_16DI_DI_Vars".DI8.xOutput,
            iFuncSystem := "SS1_750A1_16DI_DI_Vars".DI8.cFuncSystemID,
            iFuncVar := "SS1_750A1_16DI_DI_Vars".DI8.cFuncVar);
END_REGION

